Selected_Recipe_Reg_enable D270.04 BOOL  ; On if registration enabled for film
Selected_Recipe_Return_Accel D316 UINT
Selected_Recipe_Return_Decel D317 UINT
Selected_Recipe_Return_Time D314 UINT
Selected_Recipe_Return_Velocity D315 UINT
Selected_Recipe_Rev_Yank_Dist D283 UINT  ; Reverse Yank Distance
Selected_Recipe_Rewind_On_Delay D302 UINT
Selected_Recipe_Seal_Cool D300 UINT
Selected_Recipe_Seal_Delay D298 UINT
Selected_Recipe_Seal_Duration D299 UINT
Selected_Recipe_Spare_Bits_WD0_bit10 D270.10 BOOL  ; Spare
Selected_Recipe_Spare_Bits_WD0_bit11 D270.11 BOOL  ; Spare
Selected_Recipe_Spare_Bits_WD0_bit12 D270.12 BOOL  ; Spare
Selected_Recipe_Spare_Bits_WD0_bit13 D270.13 BOOL  ; Spare
Selected_Recipe_Spare_Bits_WD0_bit14 D270.14 BOOL  ; Spare
Selected_Recipe_Spare_Bits_WD0_bit15 D270.15 BOOL  ; Spare
Selected_Recipe_Spare_Bits_WD0_bit6 D270.06 BOOL  ; Spare
Selected_Recipe_Spare_Bits_WD0_bit7 D270.07 BOOL  ; Spare
Selected_Recipe_Spare_Bits_WD0_bit8 D270.08 BOOL  ; Spare
Selected_Recipe_Spare_Bits_WD0_bit9 D270.09 BOOL  ; Spare
Selected_Recipe_Spare_Bits_WD1_bit0 D271.00 BOOL  ; Spare
Selected_Recipe_Spare_Bits_WD1_bit1 D271.01 BOOL  ; Spare
Selected_Recipe_Spare_Bits_WD1_bit10 D271.10 BOOL  ; Spare
Selected_Recipe_Spare_Bits_WD1_bit11 D271.11 BOOL  ; Spare
Selected_Recipe_Spare_Bits_WD1_bit12 D271.12 BOOL  ; Spare
Selected_Recipe_Spare_Bits_WD1_bit13 D271.13 BOOL  ; Spare
Selected_Recipe_Spare_Bits_WD1_bit14 D271.14 BOOL  ; Spare
Selected_Recipe_Spare_Bits_WD1_bit15 D271.15 BOOL  ; Spare
Selected_Recipe_Spare_Bits_WD1_bit2 D271.02 BOOL  ; Spare
Selected_Recipe_Spare_Bits_WD1_bit3 D271.03 BOOL  ; Spare
Selected_Recipe_Spare_Bits_WD1_bit4 D271.04 BOOL  ; Spare
Selected_Recipe_Spare_Bits_WD1_bit5 D271.05 BOOL  ; Spare
Selected_Recipe_Spare_Bits_WD1_bit6 D271.06 BOOL  ; Spare
Selected_Recipe_Spare_Bits_WD1_bit7 D271.07 BOOL  ; Spare
Selected_Recipe_Spare_Bits_WD1_bit8 D271.08 BOOL  ; Spare
Selected_Recipe_Spare_Bits_WD1_bit9 D271.09 BOOL  ; Spare
Selected_Recipe_Spare_Bits_WD2_bit0 D272.00 BOOL  ; Spare
Selected_Recipe_Spare_Bits_WD2_bit1 D272.01 BOOL  ; Spare
Selected_Recipe_Spare_Bits_WD2_bit10 D272.10 BOOL  ; Spare
Selected_Recipe_Spare_Bits_WD2_bit11 D272.11 BOOL  ; Spare
Selected_Recipe_Spare_Bits_WD2_bit12 D272.12 BOOL  ; Spare
Selected_Recipe_Spare_Bits_WD2_bit13 D272.13 BOOL  ; Spare
Selected_Recipe_Spare_Bits_WD2_bit14 D272.14 BOOL  ; Spare
Selected_Recipe_Spare_Bits_WD2_bit15 D272.15 BOOL  ; Spare
Selected_Recipe_Spare_Bits_WD2_bit2 D272.02 BOOL  ; Spare
Selected_Recipe_Spare_Bits_WD2_bit3 D272.03 BOOL  ; Spare
Selected_Recipe_Spare_Bits_WD2_bit4 D272.04 BOOL  ; Spare
Selected_Recipe_Spare_Bits_WD2_bit5 D272.05 BOOL  ; Spare
Selected_Recipe_Spare_Bits_WD2_bit6 D272.06 BOOL  ; Spare
Selected_Recipe_Spare_Bits_WD2_bit7 D272.07 BOOL  ; Spare
Selected_Recipe_Spare_Bits_WD2_bit8 D272.08 BOOL  ; Spare
Selected_Recipe_Spare_Bits_WD2_bit9 D272.09 BOOL  ; Spare
Selected_Recipe_Spare_Bits_WD3_bit0 D273.00 BOOL  ; Spare
Selected_Recipe_Spare_Bits_WD3_bit1 D273.01 BOOL  ; Spare
Selected_Recipe_Spare_Bits_WD3_bit10 D273.10 BOOL  ; Spare
Selected_Recipe_Spare_Bits_WD3_bit11 D273.11 BOOL  ; Spare
Selected_Recipe_Spare_Bits_WD3_bit12 D273.12 BOOL  ; Spare
Selected_Recipe_Spare_Bits_WD3_bit13 D273.13 BOOL  ; Spare
Selected_Recipe_Spare_Bits_WD3_bit14 D273.14 BOOL  ; Spare
Selected_Recipe_Spare_Bits_WD3_bit15 D273.15 BOOL  ; Spare
Selected_Recipe_Spare_Bits_WD3_bit2 D273.02 BOOL  ; Spare
Selected_Recipe_Spare_Bits_WD3_bit3 D273.03 BOOL  ; Spare
Selected_Recipe_Spare_Bits_WD3_bit4 D273.04 BOOL  ; Spare
Selected_Recipe_Spare_Bits_WD3_bit5 D273.05 BOOL  ; Spare
Selected_Recipe_Spare_Bits_WD3_bit6 D273.06 BOOL  ; Spare
Selected_Recipe_Spare_Bits_WD3_bit7 D273.07 BOOL  ; Spare
Selected_Recipe_Spare_Bits_WD3_bit8 D273.08 BOOL  ; Spare
Selected_Recipe_Spare_Bits_WD3_bit9 D273.09 BOOL  ; Spare
Selected_Recipe_Spare_Bits_WD4_bit0 D274.00 BOOL  ; Spare
Selected_Recipe_Spare_Bits_WD4_bit1 D274.01 BOOL  ; Spare
Selected_Recipe_Spare_Bits_WD4_bit10 D274.10 BOOL  ; Spare
Selected_Recipe_Spare_Bits_WD4_bit11 D274.11 BOOL  ; Spare
Selected_Recipe_Spare_Bits_WD4_bit12 D274.12 BOOL  ; Spare
Selected_Recipe_Spare_Bits_WD4_bit13 D274.13 BOOL  ; Spare
Selected_Recipe_Spare_Bits_WD4_bit14 D274.14 BOOL  ; Spare
Selected_Recipe_Spare_Bits_WD4_bit15 D274.15 BOOL  ; Spare
Selected_Recipe_Spare_Bits_WD4_bit2 D274.02 BOOL  ; Spare
Selected_Recipe_Spare_Bits_WD4_bit3 D274.03 BOOL  ; Spare
Selected_Recipe_Spare_Bits_WD4_bit4 D274.04 BOOL  ; Spare
Selected_Recipe_Spare_Bits_WD4_bit5 D274.05 BOOL  ; Spare
Selected_Recipe_Spare_Bits_WD4_bit6 D274.06 BOOL  ; Spare
Selected_Recipe_Spare_Bits_WD4_bit7 D274.07 BOOL  ; Spare
Selected_Recipe_Spare_Bits_WD4_bit8 D274.08 BOOL  ; Spare
Selected_Recipe_Spare_Bits_WD4_bit9 D274.09 BOOL  ; Spare
Selected_Recipe_Spare_Bits_WD5_bit0 D275.00 BOOL  ; Spare
Selected_Recipe_Spare_Bits_WD5_bit1 D275.01 BOOL  ; Spare
Selected_Recipe_Spare_Bits_WD5_bit10 D275.10 BOOL  ; Spare
Selected_Recipe_Spare_Bits_WD5_bit11 D275.11 BOOL  ; Spare
Selected_Recipe_Spare_Bits_WD5_bit12 D275.12 BOOL  ; Spare
Selected_Recipe_Spare_Bits_WD5_bit13 D275.13 BOOL  ; Spare
Selected_Recipe_Spare_Bits_WD5_bit14 D275.14 BOOL  ; Spare
Selected_Recipe_Spare_Bits_WD5_bit15 D275.15 BOOL  ; Spare
Selected_Recipe_Spare_Bits_WD5_bit2 D275.02 BOOL  ; Spare
Selected_Recipe_Spare_Bits_WD5_bit3 D275.03 BOOL  ; Spare
Selected_Recipe_Spare_Bits_WD5_bit4 D275.04 BOOL  ; Spare
Selected_Recipe_Spare_Bits_WD5_bit5 D275.05 BOOL  ; Spare
Selected_Recipe_Spare_Bits_WD5_bit6 D275.06 BOOL  ; Spare
Selected_Recipe_Spare_Bits_WD5_bit7 D275.07 BOOL  ; Spare
Selected_Recipe_Spare_Bits_WD5_bit8 D275.08 BOOL  ; Spare
Selected_Recipe_Spare_Bits_WD5_bit9 D275.09 BOOL  ; Spare
Selected_Recipe_Spare_Bits_WD6_bit0 D276.00 BOOL  ; Spare
Selected_Recipe_Spare_Bits_WD6_bit1 D276.01 BOOL  ; Spare
Selected_Recipe_Spare_Bits_WD6_bit10 D276.10 BOOL  ; Spare
Selected_Recipe_Spare_Bits_WD6_bit11 D276.11 BOOL  ; Spare
Selected_Recipe_Spare_Bits_WD6_bit12 D276.12 BOOL  ; Spare
Selected_Recipe_Spare_Bits_WD6_bit13 D276.13 BOOL  ; Spare
Selected_Recipe_Spare_Bits_WD6_bit14 D276.14 BOOL  ; Spare
Selected_Recipe_Spare_Bits_WD6_bit15 D276.15 BOOL  ; Spare
Selected_Recipe_Spare_Bits_WD6_bit2 D276.02 BOOL  ; Spare
Selected_Recipe_Spare_Bits_WD6_bit3 D276.03 BOOL  ; Spare
Selected_Recipe_Spare_Bits_WD6_bit4 D276.04 BOOL  ; Spare
Selected_Recipe_Spare_Bits_WD6_bit5 D276.05 BOOL  ; Spare
Selected_Recipe_Spare_Bits_WD6_bit6 D276.06 BOOL  ; Spare
Selected_Recipe_Spare_Bits_WD6_bit7 D276.07 BOOL  ; Spare
Selected_Recipe_Spare_Bits_WD6_bit8 D276.08 BOOL  ; Spare
Selected_Recipe_Spare_Bits_WD6_bit9 D276.09 BOOL  ; Spare
Selected_Recipe_Spare_Bits_WD7_bit0 D277.00 BOOL  ; Spare
Selected_Recipe_Spare_Bits_WD7_bit1 D277.01 BOOL  ; Spare
Selected_Recipe_Spare_Bits_WD7_bit10 D277.10 BOOL  ; Spare
Selected_Recipe_Spare_Bits_WD7_bit11 D277.11 BOOL  ; Spare
Selected_Recipe_Spare_Bits_WD7_bit12 D277.12 BOOL  ; Spare
Selected_Recipe_Spare_Bits_WD7_bit13 D277.13 BOOL  ; Spare
Selected_Recipe_Spare_Bits_WD7_bit14 D277.14 BOOL  ; Spare
Selected_Recipe_Spare_Bits_WD7_bit15 D277.15 BOOL  ; Spare
Selected_Recipe_Spare_Bits_WD7_bit2 D277.02 BOOL  ; Spare
Selected_Recipe_Spare_Bits_WD7_bit3 D277.03 BOOL  ; Spare
Selected_Recipe_Spare_Bits_WD7_bit4 D277.04 BOOL  ; Spare
Selected_Recipe_Spare_Bits_WD7_bit5 D277.05 BOOL  ; Spare
Selected_Recipe_Spare_Bits_WD7_bit6 D277.06 BOOL  ; Spare
Selected_Recipe_Spare_Bits_WD7_bit7 D277.07 BOOL  ; Spare
Selected_Recipe_Spare_Bits_WD7_bit8 D277.08 BOOL  ; Spare
Selected_Recipe_Spare_Bits_WD7_bit9 D277.09 BOOL  ; Spare
Selected_Recipe_Spare_Bits_WD8_bit0 D278.00 BOOL  ; Spare
Selected_Recipe_Spare_Bits_WD8_bit1 D278.01 BOOL  ; Spare
Selected_Recipe_Spare_Bits_WD8_bit10 D278.10 BOOL  ; Spare
Selected_Recipe_Spare_Bits_WD8_bit11 D278.11 BOOL  ; Spare
Selected_Recipe_Spare_Bits_WD8_bit12 D278.12 BOOL  ; Spare
Selected_Recipe_Spare_Bits_WD8_bit13 D278.13 BOOL  ; Spare
Selected_Recipe_Spare_Bits_WD8_bit14 D278.14 BOOL  ; Spare
Selected_Recipe_Spare_Bits_WD8_bit15 D278.15 BOOL  ; Spare
Selected_Recipe_Spare_Bits_WD8_bit2 D278.02 BOOL  ; Spare
Selected_Recipe_Spare_Bits_WD8_bit3 D278.03 BOOL  ; Spare
Selected_Recipe_Spare_Bits_WD8_bit4 D278.04 BOOL  ; Spare
Selected_Recipe_Spare_Bits_WD8_bit5 D278.05 BOOL  ; Spare
Selected_Recipe_Spare_Bits_WD8_bit6 D278.06 BOOL  ; Spare
Selected_Recipe_Spare_Bits_WD8_bit7 D278.07 BOOL  ; Spare
Selected_Recipe_Spare_Bits_WD8_bit8 D278.08 BOOL  ; Spare
Selected_Recipe_Spare_Bits_WD8_bit9 D278.09 BOOL  ; Spare
Selected_Recipe_Spare_UINT0 D333 UINT
Selected_Recipe_Spare_UINT1 D334 UINT
Selected_Recipe_Spare_UINT10 D343 UINT
Selected_Recipe_Spare_UINT100 D433 UINT
Selected_Recipe_Spare_UINT101 D434 UINT
Selected_Recipe_Spare_UINT102 D435 UINT
Selected_Recipe_Spare_UINT103 D436 UINT
Selected_Recipe_Spare_UINT104 D437 UINT
Selected_Recipe_Spare_UINT105 D438 UINT
Selected_Recipe_Spare_UINT106 D439 UINT
Selected_Recipe_Spare_UINT107 D440 UINT
Selected_Recipe_Spare_UINT108 D441 UINT
Selected_Recipe_Spare_UINT109 D442 UINT
Selected_Recipe_Spare_UINT11 D344 UINT
Selected_Recipe_Spare_UINT110 D443 UINT
Selected_Recipe_Spare_UINT111 D444 UINT
Selected_Recipe_Spare_UINT112 D445 UINT
Selected_Recipe_Spare_UINT113 D446 UINT
Selected_Recipe_Spare_UINT114 D447 UINT
Selected_Recipe_Spare_UINT115 D448 UINT
Selected_Recipe_Spare_UINT116 D449 UINT
Selected_Recipe_Spare_UINT117 D450 UINT
Selected_Recipe_Spare_UINT118 D451 UINT
Selected_Recipe_Spare_UINT119 D452 UINT
Selected_Recipe_Spare_UINT12 D345 UINT
Selected_Recipe_Spare_UINT120 D453 UINT
Selected_Recipe_Spare_UINT121 D454 UINT
Selected_Recipe_Spare_UINT122 D455 UINT
Selected_Recipe_Spare_UINT123 D456 UINT
Selected_Recipe_Spare_UINT124 D457 UINT
Selected_Recipe_Spare_UINT125 D458 UINT
Selected_Recipe_Spare_UINT126 D459 UINT
Selected_Recipe_Spare_UINT127 D460 UINT
Selected_Recipe_Spare_UINT128 D461 UINT
Selected_Recipe_Spare_UINT129 D462 UINT
Selected_Recipe_Spare_UINT13 D346 UINT
Selected_Recipe_Spare_UINT130 D463 UINT
Selected_Recipe_Spare_UINT131 D464 UINT
Selected_Recipe_Spare_UINT132 D465 UINT
Selected_Recipe_Spare_UINT133 D466 UINT
Selected_Recipe_Spare_UINT134 D467 UINT
Selected_Recipe_Spare_UINT135 D468 UINT
Selected_Recipe_Spare_UINT136 D469 UINT
Selected_Recipe_Spare_UINT137 D470 UINT
Selected_Recipe_Spare_UINT138 D471 UINT
Selected_Recipe_Spare_UINT139 D472 UINT
Selected_Recipe_Spare_UINT14 D347 UINT
Selected_Recipe_Spare_UINT140 D473 UINT
Selected_Recipe_Spare_UINT141 D474 UINT
Selected_Recipe_Spare_UINT142 D475 UINT
Selected_Recipe_Spare_UINT143 D476 UINT
Selected_Recipe_Spare_UINT144 D477 UINT
Selected_Recipe_Spare_UINT145 D478 UINT
Selected_Recipe_Spare_UINT146 D479 UINT
Selected_Recipe_Spare_UINT147 D480 UINT
Selected_Recipe_Spare_UINT148 D481 UINT
Selected_Recipe_Spare_UINT149 D482 UINT
Selected_Recipe_Spare_UINT15 D348 UINT
Selected_Recipe_Spare_UINT150 D483 UINT
Selected_Recipe_Spare_UINT151 D484 UINT
Selected_Recipe_Spare_UINT152 D485 UINT
Selected_Recipe_Spare_UINT153 D486 UINT
Selected_Recipe_Spare_UINT154 D487 UINT
Selected_Recipe_Spare_UINT155 D488 UINT
Selected_Recipe_Spare_UINT156 D489 UINT
Selected_Recipe_Spare_UINT157 D490 UINT
Selected_Recipe_Spare_UINT158 D491 UINT
Selected_Recipe_Spare_UINT159 D492 UINT
Selected_Recipe_Spare_UINT16 D349 UINT
Selected_Recipe_Spare_UINT160 D493 UINT
Selected_Recipe_Spare_UINT161 D494 UINT
Selected_Recipe_Spare_UINT162 D495 UINT
Selected_Recipe_Spare_UINT163 D496 UINT
Selected_Recipe_Spare_UINT164 D497 UINT
Selected_Recipe_Spare_UINT165 D498 UINT
Selected_Recipe_Spare_UINT166 D499 UINT
Selected_Recipe_Spare_UINT17 D350 UINT
Selected_Recipe_Spare_UINT18 D351 UINT
Selected_Recipe_Spare_UINT19 D352 UINT
Selected_Recipe_Spare_UINT2 D335 UINT
Selected_Recipe_Spare_UINT20 D353 UINT
Selected_Recipe_Spare_UINT21 D354 UINT
Selected_Recipe_Spare_UINT22 D355 UINT
Selected_Recipe_Spare_UINT23 D356 UINT
Selected_Recipe_Spare_UINT24 D357 UINT
Selected_Recipe_Spare_UINT25 D358 UINT
Selected_Recipe_Spare_UINT26 D359 UINT
Selected_Recipe_Spare_UINT27 D360 UINT
Selected_Recipe_Spare_UINT28 D361 UINT
Selected_Recipe_Spare_UINT29 D362 UINT
Selected_Recipe_Spare_UINT3 D336 UINT
Selected_Recipe_Spare_UINT30 D363 UINT
Selected_Recipe_Spare_UINT31 D364 UINT
Selected_Recipe_Spare_UINT32 D365 UINT
Selected_Recipe_Spare_UINT33 D366 UINT
Selected_Recipe_Spare_UINT34 D367 UINT
Selected_Recipe_Spare_UINT35 D368 UINT
Selected_Recipe_Spare_UINT36 D369 UINT
Selected_Recipe_Spare_UINT37 D370 UINT
Selected_Recipe_Spare_UINT38 D371 UINT
Selected_Recipe_Spare_UINT39 D372 UINT
Selected_Recipe_Spare_UINT4 D337 UINT
Selected_Recipe_Spare_UINT40 D373 UINT
Selected_Recipe_Spare_UINT41 D374 UINT
Selected_Recipe_Spare_UINT42 D375 UINT
Selected_Recipe_Spare_UINT43 D376 UINT
Selected_Recipe_Spare_UINT44 D377 UINT
Selected_Recipe_Spare_UINT45 D378 UINT
Selected_Recipe_Spare_UINT46 D379 UINT
Selected_Recipe_Spare_UINT47 D380 UINT
Selected_Recipe_Spare_UINT48 D381 UINT
Selected_Recipe_Spare_UINT49 D382 UINT
Selected_Recipe_Spare_UINT5 D338 UINT
Selected_Recipe_Spare_UINT50 D383 UINT
Selected_Recipe_Spare_UINT51 D384 UINT
Selected_Recipe_Spare_UINT52 D385 UINT
Selected_Recipe_Spare_UINT53 D386 UINT
Selected_Recipe_Spare_UINT54 D387 UINT
Selected_Recipe_Spare_UINT55 D388 UINT
Selected_Recipe_Spare_UINT56 D389 UINT
Selected_Recipe_Spare_UINT57 D390 UINT
Selected_Recipe_Spare_UINT58 D391 UINT
Selected_Recipe_Spare_UINT59 D392 UINT
Selected_Recipe_Spare_UINT6 D339 UINT
Selected_Recipe_Spare_UINT60 D393 UINT
Selected_Recipe_Spare_UINT61 D394 UINT
Selected_Recipe_Spare_UINT62 D395 UINT
Selected_Recipe_Spare_UINT63 D396 UINT
Selected_Recipe_Spare_UINT64 D397 UINT
Selected_Recipe_Spare_UINT65 D398 UINT
Selected_Recipe_Spare_UINT66 D399 UINT
Selected_Recipe_Spare_UINT67 D400 UINT
Selected_Recipe_Spare_UINT68 D401 UINT
Selected_Recipe_Spare_UINT69 D402 UINT
Selected_Recipe_Spare_UINT7 D340 UINT
Selected_Recipe_Spare_UINT70 D403 UINT
Selected_Recipe_Spare_UINT71 D404 UINT
Selected_Recipe_Spare_UINT72 D405 UINT
Selected_Recipe_Spare_UINT73 D406 UINT
Selected_Recipe_Spare_UINT74 D407 UINT
Selected_Recipe_Spare_UINT75 D408 UINT
Selected_Recipe_Spare_UINT76 D409 UINT
Selected_Recipe_Spare_UINT77 D410 UINT
Selected_Recipe_Spare_UINT78 D411 UINT
Selected_Recipe_Spare_UINT79 D412 UINT
Selected_Recipe_Spare_UINT8 D341 UINT
Selected_Recipe_Spare_UINT80 D413 UINT
Selected_Recipe_Spare_UINT81 D414 UINT
Selected_Recipe_Spare_UINT82 D415 UINT
Selected_Recipe_Spare_UINT83 D416 UINT
Selected_Recipe_Spare_UINT84 D417 UINT
Selected_Recipe_Spare_UINT85 D418 UINT
Selected_Recipe_Spare_UINT86 D419 UINT
Selected_Recipe_Spare_UINT87 D420 UINT
Selected_Recipe_Spare_UINT88 D421 UINT
Selected_Recipe_Spare_UINT89 D422 UINT
Selected_Recipe_Spare_UINT9 D342 UINT
Selected_Recipe_Spare_UINT90 D423 UINT
Selected_Recipe_Spare_UINT91 D424 UINT
Selected_Recipe_Spare_UINT92 D425 UINT
Selected_Recipe_Spare_UINT93 D426 UINT
Selected_Recipe_Spare_UINT94 D427 UINT
Selected_Recipe_Spare_UINT95 D428 UINT
Selected_Recipe_Spare_UINT96 D429 UINT
Selected_Recipe_Spare_UINT97 D430 UINT
Selected_Recipe_Spare_UINT98 D431 UINT
Selected_Recipe_Spare_UINT99 D432 UINT
Selected_Recipe_Stale_Film_Time D329 UINT
Selected_Recipe_Temp_Setpoint D281 UINT  ; Tool temperature setpoint
Selected_Recipe_Tool_Position D319 UINT
Selected_Recipe_Top_Vacuum_Delay D286 UINT
Selected_Recipe_Tray_Position D313 UINT
Selected_Recipe_Tray_Settle_Time D307 UINT
Selected_Recipe_Tray_Stop_Delay D304 UINT
Selected_Recipe_Upstream_Off_Delay D312 UINT
Selected_Recipe_Upstream_On_Delay D311 UINT
Selected_Recipe_VAC_Type D270.00 BOOL  ; Vac type - ON = Pressure, OFF = Time
Selected_Recipe_Vacuum_Duration D288 UINT
Selected_Recipe_Vacuum_Extra_Time D290 UINT
Selected_Recipe_Vacuum_Pressure_SP D289 UINT
Selected_Recipe_Vent_Bottom_Delay D295 UINT
Selected_Recipe_Vent_Bottom_Duration D296 UINT
Selected_Recipe_Vent_Pressure_SP D297 UINT
Selected_Recipe_Vent_Top_Delay D294 UINT
Selected_Recipe_Vent_Type D270.02 BOOL  ; Vent type - ON = Pressure, OFF = Time
Servo_Drive_OK 2960.01 BOOL  ; The servo drive has no error
Servo_Drive_Reset 2961.05 BOOL  ; Reset output to servo drive
Servo_Fault W150.14 BOOL  ; Servo drive fault
Servo_Home_OK W497.01 BOOL  ; Servo home has been initiated after power up or estop condition.
Servo_On_Machine W202.15 BOOL  ; The machine has a servo drive
Simultaneous_Mode W201.04 BOOL
Sleep_Mode W151.11 BOOL  ; Sleep Mode enabled - drop temp and fault
Sleep_Mode_Delay T0220 TIMER  ; Delay to Start Sleep mode
Sleep_Mode_Minutes D898 UINT
Sleep_Mode_Temperature D899 UINT
Sleep_Mode_Temporary_Value D1142 UINT  ; Temporary register to hold the temperature setpoint while in sleep mode
Sleep_Time_SP D1140 DINT  ; Sleep timer setpoint
Slow_Down_DIstance D2400 DINT
Slow_Down_Decel H162 DINT
Slow_Down_Speed_Frequency H163 DINT  ; H163/164
Slow_Vent_Delay T0143 TIMER  ; Delay for Slow Vent
Stale_Film_timer T0215 TIMER  ; Stale film
Start_Status D800 UINT  ; Indicator status for start PB
Stepper_Pulse_Output A281.04 BOOL  ; Pulses are being output
Stop_Command W202.05 BOOL
Stop_Latch W202.04 BOOL
Stop_Status D801 UINT  ; Indicator status for stop PB
TC1_Temp_Fdbk T0150 TIMER  ; TC1 Temp Feedback Fault Delay
TC2_Temp_Fdbk T0151 TIMER  ; TC2 Temp Feedback Fault Delay
TC_AT_Enabled W501.08 BOOL  ; Set when Auto Tune is enabled
TC_Global_AT W501.06 BOOL  ; TC Global Auto Tune
TC_Loop1_AT W500.01 BOOL  ; Auto Tune Loop1
TC_Loop2_AT W500.02 BOOL  ; Auto Tune Loop2
TC_Loop3_AT W500.03 BOOL  ; Auto Tune Loop3
TC_Loop4_AT W500.04 BOOL  ; Auto Tune Loop4
TC_Loop5_AT W500.05 BOOL  ; Auto Tune Loop5
TC_Loop6_AT W500.06 BOOL  ; Auto Tune Loop6
TC_MOD1_Feedback_Fault W151.08 BOOL  ; TC Module 1 RTD Feedback Fault
TC_MOD2_Feedback_Fault W151.09 BOOL  ; TC module 2 RTD Feedback Fault
TC_PID_PROM W501.07 BOOL  ; Save PID to TC EEPROM
TC_PID_Recipe W501.10 BOOL  ; Move PID to recipe when saving
TPM D803 UINT  ; Trays Per Minute
TPO_Control_Period_Heater1 D6044 UINT  ; Time in 0.01s units of control period (200 = 2.00 seconds)
TPO_Control_Period_Heater2 D6094 UINT  ; Time in 0.01s units of control period (200 = 2.00 seconds)
TPO_Control_Period_Heater3 D6144 UINT  ; Time in 0.01s units of control period (200 = 2.00 seconds)
TPO_Control_Period_Heater4 D6194 UINT  ; Time in 0.01s units of control period (200 = 2.00 seconds)
TPO_Control_Period_Heater5 D6244 UINT  ; Time in 0.01s units of control period (200 = 2.00 seconds)
TPO_Out_Lower_Limit_Heater1 D6045 UINT  ; TPO Output lower limit when enabled in D5100.
TPO_Out_Lower_Limit_Heater2 D6095 UINT  ; TPO Output lower limit when enabled in D6043.
TPO_Out_Lower_Limit_Heater3 D6145 UINT  ; TPO Output lower limit when enabled in D6043.
TPO_Out_Lower_Limit_Heater4 D6195 UINT  ; TPO Output lower limit when enabled in D6043.
TPO_Out_Lower_Limit_Heater5 D6245 UINT  ; TPO Output lower limit when enabled in D6043.
TPO_Out_Upper_Limit_Heater1 D6046 UINT  ; TPO Output Upper limit when enabled in D5043.
TPO_Out_Upper_Limit_Heater2 D6096 UINT  ; TPO Output Upper limit when enabled in D6100.
TPO_Out_Upper_Limit_Heater3 D6146 UINT  ; TPO Output Upper limit when enabled in D6100.
TPO_Out_Upper_Limit_Heater4 D6196 UINT  ; TPO Output Upper limit when enabled in D6100.
TPO_Out_Upper_Limit_Heater5 D6246 UINT  ; TPO Output Upper limit when enabled in D6100.
TPO_Parameter1_Heater1 D6043 CHANNEL  ; Sets output limit function, input read timing, input type and MV Range
TPO_Parameter1_Heater2 D6093 CHANNEL  ; Sets output limit function, input read timing, input type and MV Range
TPO_Parameter1_Heater3 D6143 CHANNEL  ; Sets output limit function, input read timing, input type and MV Range
TPO_Parameter1_Heater4 D6193 CHANNEL  ; Sets output limit function, input read timing, input type and MV Range
TPO_Parameter1_Heater5 D6243 CHANNEL  ; Sets output limit function, input read timing, input type and MV Range
TPO_Percent_Heater1 D6042 UINT  ; Percentage output from PIDAT function
TPO_Percent_Heater2 D6092 UINT  ; Percentage output from PIDAT function
TPO_Percent_Heater3 D6142 UINT  ; Percentage output from PIDAT function
TPO_Percent_Heater4 D6192 UINT  ; Percentage output from PIDAT function
TPO_Percent_Heater5 D6242 UINT  ; Percentage output from PIDAT function
TPO_Work_Area_Word1_Heater1 D6047 CHANNEL  ; TPO Work Area - DO NOT USE FOR ANYTHING ELSE
TPO_Work_Area_Word1_Heater2 D6097 CHANNEL  ; TPO Work Area - DO NOT USE FOR ANYTHING ELSE
TPO_Work_Area_Word1_Heater3 D6147 CHANNEL  ; TPO Work Area - DO NOT USE FOR ANYTHING ELSE
TPO_Work_Area_Word1_Heater4 D6197 CHANNEL  ; TPO Work Area - DO NOT USE FOR ANYTHING ELSE
TPO_Work_Area_Word1_Heater5 D6247 CHANNEL  ; TPO Work Area - DO NOT USE FOR ANYTHING ELSE
TPO_Work_Area_Word2_Heater1 D6048 CHANNEL  ; TPO Work Area - DO NOT USE FOR ANYTHING ELSE
TPO_Work_Area_Word2_Heater2 D6098 CHANNEL  ; TPO Work Area - DO NOT USE FOR ANYTHING ELSE
TPO_Work_Area_Word2_Heater3 D6148 CHANNEL  ; TPO Work Area - DO NOT USE FOR ANYTHING ELSE
TPO_Work_Area_Word2_Heater4 D6198 CHANNEL  ; TPO Work Area - DO NOT USE FOR ANYTHING ELSE
TPO_Work_Area_Word2_Heater5 D6248 CHANNEL  ; TPO Work Area - DO NOT USE FOR ANYTHING ELSE
TPO_Work_Area_Word3_Heater1 D6049 CHANNEL  ; TPO Work Area - DO NOT USE FOR ANYTHING ELSE
TPO_Work_Area_Word3_Heater2 D6099 CHANNEL  ; TPO Work Area - DO NOT USE FOR ANYTHING ELSE
TPO_Work_Area_Word3_Heater3 D6149 CHANNEL  ; TPO Work Area - DO NOT USE FOR ANYTHING ELSE
TPO_Work_Area_Word3_Heater4 D6199 CHANNEL  ; TPO Work Area - DO NOT USE FOR ANYTHING ELSE
TPO_Work_Area_Word3_Heater5 D6249 CHANNEL  ; TPO Work Area - DO NOT USE FOR ANYTHING ELSE
Temp1_Feedback_disconnected 2009.04 BOOL  ; Input Signal Disconnected
Temp2Conv C_to_F
Temp2_Feedback_disconnected 2009.05 BOOL  ; Input Signal disconnected
Temp3Conv C_to_F
Temp4Conv C_to_F
Temp5Conv C_to_F
Temp_AutoTune_Heater1 D6009.15 BOOL  ; Initiates Autotune function
Temp_AutoTune_Heater2 D6059.15 BOOL  ; Initiates Autotune function
Temp_AutoTune_Heater3 D6109.15 BOOL  ; Initiates Autotune function
Temp_AutoTune_Heater4 D6159.15 BOOL  ; Initiates Autotune function
Temp_AutoTune_Heater5 D6209.15 BOOL  ; Initiates Autotune function
Temp_Derivative_Constant_Heater1 D6003 UINT  ; Derivative constant - 0.1s units &0 means not used
Temp_Derivative_Constant_Heater2 D6053 UINT  ; Derivative constant - 0.1s units &0 means not used
Temp_Derivative_Constant_Heater3 D6103 UINT  ; Derivative constant - 0.1s units &0 means not used
Temp_Derivative_Constant_Heater4 D6153 UINT  ; Derivative constant - 0.1s units &0 means not used
Temp_Derivative_Constant_Heater5 D6203 UINT  ; Derivative constant - 0.1s units &0 means not used
Temp_Integral_Constant_Heater1 D6002 UINT  ; Integral constant - 0.1s units.  &9999 means not used
Temp_Integral_Constant_Heater2 D6052 UINT  ; Integral constant - 0.1s units.  &9999 means not used
Temp_Integral_Constant_Heater3 D6102 UINT  ; Integral constant - 0.1s units.  &9999 means not used
Temp_Integral_Constant_Heater4 D6152 UINT  ; Integral constant - 0.1s units.  &9999 means not used
Temp_Integral_Constant_Heater5 D6202 UINT  ; Integral constant - 0.1s units.  &9999 means not used
Temp_Limit_Cycle_Hysteresis_Heater1 D6010 UINT  ; Hysteresis for limit cycle
Temp_Limit_Cycle_Hysteresis_Heater2 D6060 UINT  ; Hysteresis for limit cycle
Temp_Limit_Cycle_Hysteresis_Heater3 D6110 UINT  ; Hysteresis for limit cycle
Temp_Limit_Cycle_Hysteresis_Heater4 D6160 UINT  ; Hysteresis for limit cycle
Temp_Limit_Cycle_Hysteresis_Heater5 D6210 UINT  ; Hysteresis for limit cycle
Temp_Prop_band_Heater1 D6001 UINT  ; Proportional band in 0.1% units
Temp_Prop_band_Heater2 D6051 UINT  ; Proportional band in 0.1% units
Temp_Prop_band_Heater3 D6101 UINT  ; Proportional band in 0.1% units
Temp_Prop_band_Heater4 D6151 UINT  ; Proportional band in 0.1% units
Temp_Prop_band_Heater5 D6201 UINT  ; Proportional band in 0.1% units
Temp_Sampling_period_Heater1 D6004 UINT  ; Sampling period 0.01s units.
Temp_Sampling_period_Heater2 D6054 UINT  ; Sampling period 0.01s units.
Temp_Sampling_period_Heater3 D6104 UINT  ; Sampling period 0.01s units.
Temp_Sampling_period_Heater4 D6154 UINT  ; Sampling period 0.01s units.
Temp_Sampling_period_Heater5 D6204 UINT  ; Sampling period 0.01s units.
Temp_Set_Value_Heater1 D6000 UINT  ; Set value for the PIDAT Function
Temp_Set_Value_Heater2 D6050 UINT  ; Set value for the PIDAT Function
Temp_Set_Value_Heater3 D6100 UINT  ; Set value for the PIDAT Function
Temp_Set_Value_Heater4 D6150 UINT  ; Set value for the PIDAT Function
Temp_Set_Value_Heater5 D6200 UINT  ; Set value for the PIDAT Function
Temperature_Pressure_Scale Conv_Scale_analog_with_Int_range
Teperature_Low W150.13 BOOL  ; Temperature not high enough to run product
Termperature_High W151.07 BOOL  ; Temperature too high enough to run product
Tool_Close_Decel_Delay_Timer T0113 TIMER  ; Tool Close Delay
Tool_Down_Prox 0.03 BOOL  ; Tool down proximity sw
Tool_Down_Timer T0202 TIMER  ; Time to hold decel before releasing
Tool_Lift_Down_Decel_manual W200.05 BOOL  ; Manual tool lift down decel command
Tool_Lift_Up_Decel_manual W200.04 BOOL  ; Manual tool lift up decel command
Tool_Not_Clamped_Fault W151.04 BOOL  ; The Upper Tool Is Not Locked
Tool_Open_Decel_Delay_Timer T0112 TIMER  ; Tool Open delay
Tool_Position_HMIx10 D876 DINT
Tool_Up_Prox 0.02 BOOL  ; Tool up proximity sw
Tool_clamp_memory D967 UINT
Transducer_Fault W151.10 BOOL  ; Transducer disconnected
Tray1_AT_On_Flag 2028.03 BOOL  ; Loop1 Auto Tune ON
Tray1_ChangePIDConstants 2022.13 BOOL  ; Loop1 Turn Off PID constant flag
Tray1_Constants_Calculated 2028.10 BOOL  ; Loop1 PID Constants Calc flag
Tray1_ControlPeriod_SP D20213 UINT
Tray1_Derivative D20217 UINT
Tray1_FATALCONTROL_Error 2028.12 BOOL  ; Loop1 FATAL CONTROL Error
Tray1_Integral_Time D20216 UINT
Tray1_Output_On 2028.04 BOOL  ; Loop1 Control Output ON
Tray1_PID_Save 2022.15 BOOL  ; Loop1 Save to EEPROM
Tray1_PV 2023 INT  ; Loop1 Process Value
Tray1_Proportional D20215 UINT
Tray1_SENSOR_Error 2028.14 BOOL  ; Loop1 SENSOR error
Tray1_SETTING_Error 2028.09 BOOL  ; Loop1 SETTING Error
Tray1_SP 2020 INT  ; Loop1 Setpoint
Tray1_Save_Complete 2028.15 BOOL  ; Loop1 Save to EEPROM complete
Tray1_Start_AT 2022.02 BOOL  ; Loop1 Start Auto Tune
Tray1_Stop 2022.06 BOOL  ; Loop1 Stop Controlling
Tray1_StopAT 2022.03 BOOL  ; Loop1 Stop Auto Tune
Tray1_Stop_Sensor 1.00 BOOL  ; Tray stop sensor input
Tray1_Temp_Fdbk T0145 TIMER  ; Tray 1 Temp Feedback Fault Delay
Tray1and2_Alarm_Mode D20200 CHANNEL
Tray2_AT_On_Flag 2029.03 BOOL  ; Loop2 Auto Tune ON
Tray2_ChangePIDConstants 2022.12 BOOL  ; Loop2 Turn Off PID constant flag
Tray2_Constants_Calculated 2029.10 BOOL  ; Loop2 PID Constants Calc flag
Tray2_ControlPeriod_SP D20223 UINT
Tray2_Derivative D20227 UINT
Tray2_FATALCONTROL_Error 2029.12 BOOL  ; Loop2 FATAL CONTROL Error
Tray2_Integral_Time D20226 UINT
Tray2_Output_On 2029.04 BOOL  ; Loop2 Control Output ON
Tray2_PID_Save 2022.14 BOOL  ; Loop2 Save to EEPROM
Tray2_PV 2024 INT  ; Loop2 Process Value
Tray2_Proportional D20225 UINT
Tray2_SENSOR_Error 2029.14 BOOL  ; Loop2 SENSOR error
Tray2_SETTING_Error 2029.09 BOOL  ; Loop2 SETTING Error
Tray2_SP 2021 INT  ; Loop2 Setpoint
Tray2_Save_Complete 2029.15 BOOL  ; Loop2 Save to EEPROM complete
Tray2_Start_AT 2022.00 BOOL  ; Loop2 Start Auto Tune
Tray2_Stop 2022.04 BOOL  ; Loop2 Stop Controlling
Tray2_Stop_AT 2022.01 BOOL  ; Loop2 Stop Auto Tune
Tray2_Stop_Sensor 1.01 BOOL  ; Tray stop sensor input
Tray2_Temp_Fdbk T0146 TIMER  ; Tray 2 Temp Feedback Fault Delay
Tray3_AT_On_Flag 2038.03 BOOL  ; Loop3 Auto Tune ON
Tray3_ChangePIDConstants 2032.13 BOOL  ; Loop3 Turn Off PID constant flag
Tray3_Constants_Calculated 2038.10 BOOL  ; Loop3 PID Constants Calc flag
Tray3_ControlPeriod_SP D20253 UINT
Tray3_Derivative D20257 UINT
Tray3_FATALCONTROL_Error 2038.12 BOOL  ; Loop3 FATAL CONTROL Error
Tray3_Integral_Time D20256 UINT
Tray3_Output_On 2038.04 BOOL  ; Loop3 Control Output ON
Tray3_PID_Save 2032.15 BOOL  ; Loop3 Save to EEPROM
Tray3_PV 2033 INT  ; Loop3 Process Value
Tray3_Proportional D20255 UINT
Tray3_SENSOR_Error 2038.14 BOOL  ; Loop3 SENSOR error
Tray3_SETTING_Error 2038.09 BOOL  ; Loop3 SETTING Error
Tray3_SP 2030 INT  ; Loop 3 Setpoint
Tray3_Save_Complete 2038.15 BOOL  ; Loop3 Save to EEPROM complete
Tray3_Start_AT 2032.02 BOOL  ; Loop3 Start Auto Tune
Tray3_Stop 2032.06 BOOL  ; Loop3 Stop Controlling
Tray3_Stop_AT 2032.03 BOOL  ; Loop3 Stop Auto Tune
Tray3_Stop_Sensor 1.02 BOOL  ; Tray stop sensor input
Tray3_Temp_Fdbk T0147 TIMER  ; Tray 3 Temp Feedback Fault Delay
Tray3and4_Alarm_Mode D20201 CHANNEL
Tray4_AT_On_Flag 2039.03 BOOL  ; Loop4 Auto Tune ON
Tray4_ChangePIDConstants 2032.12 BOOL  ; Loop4 Turn Off PID constant flag
Tray4_Constants_Calculated 2039.10 BOOL  ; Loop4 PID Constants Calc flag
Tray4_ControlPeriod_SP D20263 UINT
Tray4_Derivative D20267 UINT
Tray4_FATALCONTROL_Error 2039.12 BOOL  ; Loop4 FATAL CONTROL Error
Tray4_Integral_Time D20266 UINT
Tray4_Output_On 2039.04 BOOL  ; Loop4 Control Output ON
Tray4_PID_Save 2032.14 BOOL  ; Loop4 Save to EEPROM
Tray4_PV 2034 INT  ; Loop4 Process Value
Tray4_Proportional D20265 UINT
Tray4_SENSOR_Error 2039.14 BOOL  ; Loop4 SENSOR error
Tray4_SETTING_Error 2039.09 BOOL  ; Loop4 SETTING Error
Tray4_SP 2031 INT  ; Loop 4 Setpoint
Tray4_Save_Complete 2039.15 BOOL  ; Loop4 Save to EEPROM complete
Tray4_Start_AT 2032.00 BOOL  ; Loop4 Start Auto Tune
Tray4_Stop 2032.04 BOOL  ; Loop4 Stop Controlling
Tray4_Stop_AT 2032.01 BOOL  ; Loop4 Stop Auto Tune
Tray4_Stop_Sensor 1.03 BOOL  ; Tray stop sensor input
Tray4_Temp_Fdbk T0148 TIMER  ; Tray 4 Temp Feedback Fault Delay
Tray5_AT_On_Flag 2128.03 BOOL  ; Loop5 Auto Tune ON
Tray5_ChangePIDConstants 2122.13 BOOL  ; Loop5 Turn Off PID constant flag
Tray5_Constants_Calculated 2128.10 BOOL  ; Loop5 PID Constants Calc flag
Tray5_ControlPeriod_SP D21213 UINT
Tray5_Derivative D21217 UINT
Tray5_FATALCONTROL_Error 2128.12 BOOL  ; Loop5 FATAL CONTROL Error
Tray5_Integral_Time D21216 UINT
Tray5_Output_On 2128.04 BOOL  ; Loop5 Control Output ON
Tray5_PID_Save 2122.15 BOOL  ; Loop5 Save to EEPROM
Tray5_PV 2123 INT  ; Loop5 Process Value
Tray5_Proportional D21215 UINT
Tray5_SENSOR_Error 2128.14 BOOL  ; Loop5 SENSOR error
Tray5_SETTING_Error 2128.09 BOOL  ; Loop5 SETTING Error
Tray5_SP 2120 INT  ; Loop 5 Setpoint
Tray5_Save_Complete 2128.15 BOOL  ; Loop5 Save to EEPROM complete
Tray5_Start_AT 2122.02 BOOL  ; Loop5 Start Auto Tune
Tray5_Stop 2122.06 BOOL  ; Loop5 Stop Controlling
Tray5_StopAT 2122.03 BOOL  ; Loop5 Stop Auto Tune
Tray5_Stop_Sensor 1.04 BOOL  ; Tray stop sensor input
Tray5_Temp_Fdbk T0149 TIMER  ; Tray 5 Temp Feedback Fault Delay
Tray5and6_Alarm_Mode D21200 CHANNEL
Tray6_ControlPeriod_SP D21223 UINT
Tray6_Derivative D21227 UINT
Tray6_Integral_Time D21226 UINT
Tray6_Proportional D21225 UINT
TrayCountChanged W203.08 BOOL  ; The tray count has been changed.
TrayStop1_Off_Filter_Timer T0262 TIMER
TrayStop2_Off_Filter_Timer T0263 TIMER
TrayStop3_Off_Filter_Timer T0264 TIMER
TrayStop4_Off_Filter_Timer T0265 TIMER
TrayStop5_Off_Filter_Timer T0266 TIMER
TrayStop6_Off_Filter_Timer T0267 TIMER
Tray_Count D512 UINT  ; Trays past the infeed gate
Tray_Detected_4_measurement 1.09 BOOL  ; Photocell to detect trays for measurement
Tray_Height_Int D2026 UINT  ; Tray height in INT form
Tray_Height_memory1 D2027 UINT  ; Measured hieght of tray 1
Tray_Height_memory2 D2028 UINT  ; Measured height of tray2
Tray_Height_memory3 D2029 UINT  ; Measured height of tray3
Tray_Height_memory4 D2030 UINT  ; Measured height of tray4
Tray_Height_memory5 D2031 UINT  ; Measured height of tray5
Tray_Measured T0242 TIMER  ; Measured Time for tray passage
Tray_Measurement_bits D2034 UINT  ; Bits used for tray measurement
Tray_Measurement_counter D2033 UINT  ; Measurement counter
Tray_Position_HMIx10 D878 DINT
Tray_count_TPM D965 UINT
Tray_filter T0253 TIMER  ; Filter signal for tray counting
Tray_measure_delay T0251 TIMER  ; Delay tray measurement
Tray_measurement_bits D2034.00 BOOL  ; Meaurement in progress
Tray_measurement_temp D2032 UINT  ; temporary memory location for tray height
Tray_measurement_timer T0252 TIMER  ; Time to measure tray
UPPER_TOOL_UNLOCK_DELAY T0126 TIMER  ; Delay Upper Tool from Unlocking
UnitRestart_TC102_1 A502.02 BOOL  ; Restart TC102 Module 1
UnitRestart_TC102_2 A502.12 BOOL  ; Restart TC102 Module 2
UpStream_Conv_Timer_Input T0224 TIMER  ; UpStream_Conv_Timer_Input_HMI
UpStream_Conv_photo_Eye 1.08 BOOL  ; UpStream Conv. Photo-Eye
UpperTool_Unlocked_Status H100.00 BOOL
Upper_Tool_DN_EStop W203.12 BOOL  ; Send Upper Tool Down if E-Stop hit during Lock motion
Upper_Tool_Feedback_NOP W203.14 BOOL
Upper_Tool_Jammed W153.13 BOOL  ; Upper Tool Jammed while trying to close
Upper_Tool_Lock_WD_Fault W150.06 BOOL  ; Watchdog Timer Fault
Upper_Tool_Lock_WD_Timer T0135 TIMER  ; Watchdog Timer
Upper_Tool_Locked W203.09 BOOL  ; Upper Tool Locked when a Safety Faults
Upper_Tool_NOT_Locked W203.11 BOOL  ; Upper Tool NOT Locked Bit
Upper_Tool_Pressure 2005 UINT  ; Upper Tool Pressure
Upper_Tool_Temp_IN5 2017 UINT
Upper_Tool_UNLocked W203.10 BOOL  ; Upper Tool UnLocked when a Safety Trips
Upper_Tool_Unlock_WD_Fault W150.07 BOOL  ; Watchdog Timer Fault
Upper_Tool_Unlock_WD_Timer T0136 TIMER  ; Watchdog Timer
Upper_Tool_Unlocked H100.00 BOOL  ; Upper Tool unlocked status
Upper_Tool_Up_Request W203.13 BOOL  ; HMI Tool Up/Lock Pressed
Upper_Vac_Duration_Simultaneous_Timer T0208 TIMER  ; Used for simultaneous Mode
Upstream_Off_Timer T0210 TIMER  ; OFF Delay timer for upstream signal
Upstream_On_Timer T0209 TIMER  ; ON Delay timer for upstream signal
V10_Tray_2_Stop_Extend 3.09 BOOL  ; V10 Tray Stop 2 Extend output
V11_Tray_Stop3_Extend 4.03 BOOL  ; V11 Tray Stop 3 Extend output
V12_Tray_Stop4_Extend 4.04 BOOL  ; V12 Tray Stop 4 Extend output
V13_Tray_Stop5_Extend 4.05 BOOL  ; V13 Tray Stop 5 Extend output
V14_Infeed_Gate_Retract 3.04 BOOL  ; V14 Infeed Gate Retract output
V15A_Seal_Bar_Retract 2.06 BOOL  ; V15A Seal Bar Retract output
V15B_Seal_Bars_Extend 2.07 BOOL  ; V15B Seal Bar Extend output
V16A_Lower_Tool_Up 2.14 BOOL  ; V16A Lower Tool Lift Up output
V16B_Lower_Tool_Dn 2.15 BOOL  ; V16B Lower Tool Lift Down output
V17A_Lower_Tool_Up_Decel 3.00 BOOL  ; V17A Lower Tool Decel for Up movement
V17B_Lower_Tool_Dn_Decel 3.01 BOOL  ; V17B Lower Tool Decel for Down movement
V1A_Upper_Tool_Vac 2.09 BOOL  ; V1A Upper Tool Vac On output
V1B_Upper_Tool_Vent_Close 2.10 BOOL  ; V1B Upper Tool Vent Close output
V2A_Lower_Tool_Vac 2.11 BOOL  ; V2A Lower Tool Vacuum On output
V2B_Lower_Tool_Vent_Close 2.12 BOOL  ; V2B Vent Close On output
V33_Upstream_Tray_Stop 3.13 BOOL  ; V33 Upstream_Conv_Tray_Stop
V4A_Gripper_Close 3.02 BOOL  ; V4A Tray Gripper Close output
V4B_Gripper_Open 3.03 BOOL  ; V4B Tray Gripper Open output
V5A_Gas_On 2.13 BOOL  ; V5A Gas ON output
V5B_Slow_Top_Vent 3.12 BOOL  ; V5B Slow Top Vent -Option
V6A_Upper_Tool_UnLock 2.03 BOOL  ; V6A Unlock Upper Tool Seat
V6B_Upper_Tool_Lock 3.11 BOOL  ; V6B Lock/Raise Upper Tool-double solenoid valve only
V7_Lower_Tool_Center_Seal 2.04 BOOL  ; V7 Lower Tool Center Seal On
V8A_Gripper_Extend 3.05 BOOL  ; V8A Gripper Extend output-IN450 ONLY
V8B_Gripper_Retract 3.06 BOOL  ; V8B Gripper Retract output-IN450 ONLY
V9_Tray_1_Stop_Extend 3.08 BOOL  ; V9 Tray 1 Stop 1 Extend output
VSP_Mode W201.05 BOOL
VacGraph_Pause W503.02 BOOL  ; graph pause
Vac_Delay_Timer_Bottom T0115 TIMER  ; Vacuum delay timer -Bottom Valve
Vac_Delay_Timer_Top T0114 TIMER  ; Vacuum delay timer - Top Valve
Vac_Duration_Timer T0116 TIMER  ; Vacuum duration
Vac_Test1 Vac_Test_Calc
Vac_Test_Cycle_Timer T0218 TIMER  ; Allowable time for cycle
Vac_Test_Leak_Time D1138 CHANNEL  ; Time for pressure to leak off
Vac_Test_Leak_reached W202.03 BOOL  ; The leak pressure has been reached.
Vac_Test_Pressure_Reached W202.02 BOOL  ; Vacuum test pressure reached
Vac_Test_Result_Time D1137 UINT  ; Time to draw vacuum
Vac_Test_Vent_Timer T0217 TIMER  ; Vent timer release for vacuum test
Vac_Test_ended_early W202.07 BOOL  ; Vac test ended early
Vac_Timeout_WD_Fault W150.05 BOOL  ; Watchdog Timer Fault
Vac_Timeout_WD_Timer T0134 TIMER  ; Watchdog Timer
Vacuum_Extra_time T0219 TIMER
Vacuum_Pump_OK 0.14 BOOL  ; Vacuum pump OK input
Vacuum_Test_Fault W151.06 BOOL
Vacuum_Test_Finished W203.05 BOOL  ; Vacuum test completely finished
Vacuum_Test_Status D960 UINT
Vent_Delay_Timer_Bottom T0120 TIMER  ; Vent Delay Timer - Bottom Valve
Vent_Delay_Timer_Top T0119 TIMER  ; Vent Delay Timer - Top Valve
Vent_Duration_Timer T0121 TIMER  ; Vent duration Timer
Vent_Timeout_WD_Fault W150.10 BOOL  ; Watchdog Timer Fault
Vent_Timeout_WD_Timer T0139 TIMER  ; Watchdog Timer
Vx_UpStream_Tray_Stop_Extend 4.06 BOOL  ; Vx Upstream Conveyor Tray Stop Extend
Yank_Accel_Rate H20 UINT
Yank_Decel_Rate H21 UINT
Yank_Distance_Negative D1114 DINT
Yank_Starting_Freq H26 DINT
Yank_Target_Frequency H22 DINT
Yank_Target_Position H24 DINT
aiCard2_Channel4 2018 UINT
aiForceEnable_Card1Channel4 D2010.05 BOOL  ; unused
aiForceEnable_UpperToolTemp1 D2010.02 BOOL  ; Temperature input1 upper tool force enable
aiForceEnable_UpperToolTemp2 D2010.03 BOOL  ; Temperature input2 upper tool force enable
aiForceEnable_VacuumPressure D2010.04 BOOL  ; pressure transducer for upper tool force enable
aiValue_Card1Channel4 D2025 UINT  ; unused
aiValue_UpperToolTemp1 D2022 UINT  ; Temperature input1 upper tool logical value
aiValue_UpperToolTemp2 D2023 UINT  ; Temperature input2 upper tool logical value
aiValue_VacuumPressure D2024 UINT  ; pressure transducer for upper tool logical value
aoForceEnable_Card1Channel2 D2010.01 BOOL  ; One shot for Measure
aoForceEnable_InfeedConveyorSpeedRef D2010.00 BOOL  ; Analog output for speed reference force enable
aoValue_Card1Channel2 D2021 UINT  ; unused
aoValue_InfeedConveyorSpeedRef D2020 UINT  ; Analog output for speed reference logical value
bActivateSealBarHeating D5053.00 BOOL
bEnglishMode D910.00 BOOL
bFaultOverTemperature D5053.01 BOOL
bFaultTemperatureDeviation D5053.02 BOOL
bGripperJogCommanded D5053.09 BOOL  ; jog button pressed on HMI
bGripperJogging D5053.10 BOOL  ; gripper in jog sequence
bSetTempControlParameters D5053.04 BOOL
bTunePID D5053.03 BOOL
cfgAi1MeanSampleSetting D20006 CHANNEL  ; set to 16 samples for mean
cfgAi2MeanSampleSetting D20007 CHANNEL  ; set to 16 samples for mean
cfgAi3MeanSampleSetting D20008 CHANNEL  ; set to 8 samples for mean
cfgAi4MeanSampleSetting D20009 CHANNEL  ; set to 8 samples for mean
gas_rescale_result D2045 WORD
iGripperJogStep D5500 UINT
iTempDeviationHolder D5055 UINT
iTempDeviationHolder1 D5057 UINT
ipCard2Bit10 1.10 BOOL  ; unused
ipForceEnable_ACDrive_OK D2002.07 BOOL  ; AC Drive Input Force enable
ipForceEnable_AirPressureOk D2000.04 BOOL  ; Air Pressure switch Force enable
ipForceEnable_FrontGrippedClosed D2000.07 BOOL  ; Front Gripper closed proximity sw Force enable
ipForceEnable_FrontGripperOpen D2000.06 BOOL  ; Front Gripper open proximity switch Force enable
ipForceEnable_GasPressureOk D2000.05 BOOL  ; Gas Pressure Switch Force enable
ipForceEnable_GripperExtended D2000.08 BOOL  ; Gripper extended proximity sw Force enable
ipForceEnable_GripperRetracted D2000.09 BOOL  ; Gripper retracted proximity sw Force enable
ipForceEnable_GuardAuthority D2000.15 BOOL  ; Guard Authority input Force enable
ipForceEnable_GuardOk D2000.11 BOOL  ; Guard door switches ok Force enable
ipForceEnable_InfeedEstop D2000.01 BOOL  ; E-Stop circuit status Force enable
ipForceEnable_InfeedGate D2000.12 BOOL  ; Infeed Gate Sensor Force enable
ipForceEnable_OutfeedEstop D2000.10 BOOL  ; E-Stop circuit status Force enable
ipForceEnable_Rear_Gripper_Closed_Prox D2002.06 BOOL  ; Rear Gripper closed prox Force Enable
ipForceEnable_Rear_Gripper_Open_Prox D2002.05 BOOL  ; Rear Gripper Open prox Force Enable
ipForceEnable_RemotePause D2000.13 BOOL  ; Remote pause input Force enable
ipForceEnable_RewindDancerUp D2000.00 BOOL  ; Proximity sw input Force enable
ipForceEnable_StopSensorTray1 D2002.00 BOOL  ; Tray stop sensor input Force enable
ipForceEnable_StopSensorTray2 D2002.01 BOOL  ; Tray stop sensor input Force enable
ipForceEnable_StopSensorTray3 D2002.02 BOOL  ; Tray stop sensor input Force enable
ipForceEnable_StopSensorTray4 D2002.03 BOOL  ; Tray stop sensor input Force enable
ipForceEnable_StopSensorTray5 D2002.04 BOOL  ; Tray stop sensor input Force enable
ipForceEnable_ToolDown D2000.03 BOOL  ; Tool down proximity sw Force enable
ipForceEnable_ToolUp D2000.02 BOOL  ; Tool up proximity sw Force enable
ipForceEnable_VacuumPumpOk D2000.14 BOOL  ; Vacuum pump OK input Force enable
ipForceEnable_ipCard2Bit10 D2002.10 BOOL  ; unused Force enable
ipForceEnable_ipCard2Bit11 D2002.11 BOOL  ; unused Force enable
ipForceEnable_ipCard2Bit12 D2002.12 BOOL  ; unused Force enable
ipForceEnable_ipCard2Bit13 D2002.13 BOOL  ; unused Force enable
ipForceEnable_ipCard2Bit14 D2002.14 BOOL  ; unused Force enable
ipForceEnable_ipCard2Bit15 D2002.15 BOOL  ; unused Force enable
ipForceEnable_ipCard2Bit7 D2002.07 BOOL  ; unused Force enable
ipForceEnable_ipCard2Bit8 D2002.08 BOOL  ; unused Force enable
ipForceEnable_ipCard2Bit9 D2002.09 BOOL  ; unused Force enable
ipState_AC_Drive_OK D2003.07 BOOL  ; AC Drive OK input logical State
ipState_AirPressureOk D2001.04 BOOL  ; Air Pressure switch logical State
ipState_FrontGrippedClosed D2001.07 BOOL  ; Front Gripper closed proximity sw logical State
ipState_FrontGripperOpen D2001.06 BOOL  ; Front Gripper open proximity switch logical State
ipState_GasPressureOk D2001.05 BOOL  ; Gas Pressure Switch logical State
ipState_GripperExtended D2001.08 BOOL  ; Gripper extended proximity sw logical State
ipState_GripperRetracted D2001.09 BOOL  ; Gripper retracted proximity sw logical State
ipState_GuardAuthority D2001.15 BOOL  ; Guard Authority input logical State
ipState_GuardOk D2001.11 BOOL  ; Guard door switches ok logical State
ipState_InfeedEstop D2001.01 BOOL  ; E-Stop circuit status logical State
ipState_InfeedGate D2001.12 BOOL  ; Infeed Gate Sensor logical State
ipState_OutfeedEstop D2001.10 BOOL  ; E-Stop circuit status logical State
ipState_Printer_Fault D2003.15 BOOL  ; Bell-Mark Printer
ipState_Printer_Ready D2003.14 BOOL  ; Bell-Mark Printer
ipState_Rear_Gripper_Closed_Prox D2003.06 BOOL  ; Rear gripper closed logical state
ipState_Rear_Gripper_Open_Prox D2003.05 BOOL  ; Rear gripper Open logical state
ipState_RemotePause D2001.13 BOOL  ; Remote pause input logical State
ipState_RewindDancerUp D2001.00 BOOL  ; Proximity sw input logical State
ipState_StopSensorTray1 D2003.00 BOOL  ; Tray stop sensor input logical State
ipState_StopSensorTray2 D2003.01 BOOL  ; Tray stop sensor input logical State
ipState_StopSensorTray3 D2003.02 BOOL  ; Tray stop sensor input logical State
ipState_StopSensorTray4 D2003.03 BOOL  ; Tray stop sensor input logical State
ipState_StopSensorTray5 D2003.04 BOOL  ; Tray stop sensor input logical State
ipState_ToolDown D2001.03 BOOL  ; Tool down proximity sw logical State
ipState_ToolUp D2001.02 BOOL  ; Tool up proximity sw logical State
ipState_UpStream_PE D2003.08 BOOL  ; UpStream_Photo_Eye
ipState_VacuumPumpOk D2001.14 BOOL  ; Vacuum pump OK input logical State
ipState_ipCard2Bit10 D2003.10 BOOL  ; unused logical State
ipState_ipCard2Bit11 D2003.11 BOOL  ; Infeed safety door
ipState_ipCard2Bit12 D2003.12 BOOL  ; Front or Back Door Safety
ipState_ipCard2Bit13 D2003.13 BOOL
ipState_ipCard2Bit9 D2003.09 BOOL  ; unused logical State
keyswitch_Input_Access 1.12 BOOL  ; Keyswitc input for access to parameters
opCard2Bit14 3.14 BOOL  ; unused
opCard3Bit10 4.10 BOOL  ; unused
opCard3Bit11 4.11 BOOL  ; unused
opCard3Bit12 4.12 BOOL  ; unused
opCard3Bit13 4.13 BOOL  ; unused
opCard3Bit7 4.07 BOOL  ; unused
opCard3Bit8 4.08 BOOL  ; unused
opCard3Bit9 4.09 BOOL  ; unused
opForceEnable_Card2Bit12 D2006.12 BOOL  ; unused Force enable
opForceEnable_Card2Bit13 D2006.13 BOOL  ; unused Force enable
opForceEnable_Card2Bit14 D2006.14 BOOL  ; unused Force enable
opForceEnable_Card2Bit15 D2006.15 BOOL  ; unused Force enable
opForceEnable_Card3Bit10 D2008.10 BOOL  ; unused Force enable
opForceEnable_Card3Bit11 D2008.11 BOOL  ; unused Force enable
opForceEnable_Card3Bit12 D2008.12 BOOL  ; unused Force enable
opForceEnable_Card3Bit13 D2008.13 BOOL  ; unused Force enable
opForceEnable_Card3Bit7 D2008.07 BOOL  ; unused Force enable
opForceEnable_Card3Bit8 D2008.08 BOOL  ; unused Force enable
opForceEnable_Card3Bit9 D2008.09 BOOL  ; unused Force enable
opForceEnable_GasOn D2004.13 BOOL  ; Gas ON output Force enable
opForceEnable_GripperExtend D2006.05 BOOL  ; Gripper Extend output Force enable
opForceEnable_GripperRetract D2006.06 BOOL  ; Gripper Retract output Force enable
opForceEnable_HeatCR D2004.00 BOOL  ; Heat contactor output Force enable
opForceEnable_InfeedConveyorRun D2006.07 BOOL  ; Run the infeed conveyor Force enable
opForceEnable_InfeedGateRetract D2006.04 BOOL  ; Infeed gate retract output Force enable
opForceEnable_LowerToolLiftDown D2004.15 BOOL  ; Lower tool lift down output Force enable
opForceEnable_LowerToolLiftDownDecel D2006.01 BOOL  ; Tool Decel output for down movement Force enable
opForceEnable_LowerToolLiftUp D2004.14 BOOL  ; Lower tool lift up output Force enable
opForceEnable_LowerToolLiftUpDecel D2006.00 BOOL  ; Tool Decel output for up movement Force enable
opForceEnable_LowerToolVac D2004.11 BOOL  ; Lower tool vacuum output Force enable
opForceEnable_LowerToolVentClose D2004.12 BOOL  ; Vent close output Force enable
opForceEnable_Printer_Enable D2008.14 BOOL  ; Bell-Mark Printer
opForceEnable_Printer_Print D2008.15 BOOL  ; Bell-Mark Printer
opForceEnable_RewindMotorStarter D2004.08 BOOL  ; Rewind Motor output Force enable
opForceEnable_SealBarExtend D2004.07 BOOL  ; Seal bars extend output Force enable
opForceEnable_SealBarHeat D2004.01 BOOL  ; Seal Bar Heat output Force enable
opForceEnable_SealBarHeat_2 D2004.02 BOOL  ; Seal Bar Heat output logical State Heater 2
opForceEnable_SealBarRetract D2004.06 BOOL  ; Seal bar retract output Force enable
opForceEnable_Seal_Bar_Heat_3 D2008.00 BOOL  ; Seal Bar Heat output 3 Force Enable
opForceEnable_Seal_Bar_Heat_4 D2008.01 BOOL  ; Seal Bar Heat output 4 Force Enable
opForceEnable_Seal_Bar_Heat_5 D2008.02 BOOL  ; Seal Bar Heat output 5 Force Enable
opForceEnable_TrayGripClose D2006.02 BOOL  ; Grip close output Force enable
opForceEnable_TrayGripOpen D2006.03 BOOL  ; Grip open output Force enable
opForceEnable_TrayStop1Extend D2006.08 BOOL  ; Tray stop 1 extend output Force enable
opForceEnable_TrayStop2Extend D2006.09 BOOL  ; Tray stop 2 extend output Force enable
opForceEnable_Tray_Stop3_Extend D2008.03 BOOL  ; Tray stop 3 extend output Force Enable
opForceEnable_Tray_Stop4_Extend D2008.04 BOOL  ; Tray stop 4 extend output Force Enable
opForceEnable_Tray_Stop5_Extend D2008.05 BOOL  ; Tray stop 5 extend output Force Enable
opForceEnable_UpperToolVac D2004.09 BOOL  ; Upper tool vacuum output Force enable
opForceEnable_UpperToolVentClose D2004.10 BOOL  ; Upper tool vent close output Force enable
opForceEnable_UpstreamStop D2006.10 BOOL  ; Upstream Stop output Force enable
opForceEnable_V6A_UpperToolSeat D2004.03 BOOL  ; V6A Upper Tool Seat UNLock Force enable
opForceEnable_V6B_UpperTool_Lock D2006.11 BOOL  ; Upper Tool Lock Output Force enable
opForceEnable_V7_LowerToolSeal D2004.04 BOOL  ; V7 Lower tool Center Seal output Force enable
opForceEnable_VacuumPump D2004.05 BOOL  ; Vacuum Pump output Force enable
opForceState_V6UpperToolSeat W102.05 BOOL  ; used to force Upper Tool seat output
opForceUpstream_Stop D2008.06 BOOL  ; Force Enable for upstream stop
opState_Card2Bit14 D2007.14 BOOL  ; unused logical State
opState_Force_Tool_Decel_Down D2009.08 BOOL  ; Force Decel Down Immediately
opState_GasOn D2005.13 BOOL  ; Gas ON output logical State
opState_GripperExtend D2007.05 BOOL  ; Gripper Extend output logical State
opState_GripperRetract D2007.06 BOOL  ; Gripper Retract output logical State
opState_HeatCR D2005.00 BOOL  ; Heat contactor output logical State
opState_InfeedConveyorRun D2007.07 BOOL  ; Run the infeed conveyor logical State
opState_InfeedGateRetract D2007.04 BOOL  ; Infeed gate retract output logical State
opState_Lift_Up_B4_lowering D2009.09 BOOL  ; Reenergize Lift before lowering
opState_LowerToolLiftDown D2005.15 BOOL  ; Lower tool lift down output logical State
opState_LowerToolLiftDownDecel D2007.01 BOOL  ; Tool Decel output for down movement logical State
opState_LowerToolLiftUp D2005.14 BOOL  ; Lower tool lift up output logical State
opState_LowerToolLiftUpDecel D2007.00 BOOL  ; Tool Decel output for up movement logical State
opState_LowerToolVac D2005.11 BOOL  ; Lower tool vacuum output logical State
opState_LowerToolVentClose D2005.12 BOOL  ; Vent close output logical State
opState_Outfeed_Conveyor D2007.15 BOOL  ; Run outfeed conveyor
opState_Printer_Enable D2009.14 BOOL  ; Bell-Mark Printer
opState_Printer_Print D2009.15 BOOL  ; Bell-Mark Printer
opState_Renergize_button D2009.10 BOOL  ; HMI open and exit button
opState_RewindMotorStarter D2005.08 BOOL  ; Rewind Motor output logical State
opState_SealBar1_Heat D2005.01 BOOL  ; Seal Bar 1 Heat output logical State
opState_SealBarExtend D2005.07 BOOL  ; Seal bars extend output logical State
opState_SealBarRetract D2005.06 BOOL  ; Seal bar retract output logical State
opState_Seal_Bar_Heat_3 D2009.00 BOOL  ; Seal Bar Heat output 3
opState_Seal_Bar_Heat_4 D2009.01 BOOL  ; Seal Bar Heat output 4
opState_Seal_Bar_Heat_5 D2009.02 BOOL  ; Seal Bar Heat output 5
opState_Sealbar2_heat D2005.02 BOOL  ; Heat output for seal bar 2
opState_TrayGripClose D2007.02 BOOL  ; Grip close output logical State
opState_TrayGripOpen D2007.03 BOOL  ; Grip open output logical State
opState_TrayStop1Extend D2007.08 BOOL  ; Tray stop 1 extend output logical State
opState_TrayStop2Extend D2007.09 BOOL  ; Tray stop 2 extend output logical State
opState_TrayStop3Extend D2009.03 BOOL  ; Extend Tray stop 3
opState_TrayStop4Extend D2009.04 BOOL  ; Extend tray stop 4
opState_TrayStop5Extend D2009.05 BOOL  ; Extend tray stop 5
opState_UpperToolVac D2005.09 BOOL  ; Upper tool vacuum output logical State
opState_UpperToolVentClose D2005.10 BOOL  ; Upper tool vent close output logical State
opState_UpstreamStop D2007.10 BOOL  ; Upstream Stop output logical State
opState_Upstream_Stop_Bit_2 D2009.07 BOOL  ; Upstream Stop bit
opState_V33_Upstream_Stop D2007.13 BOOL  ; V33 Upstream Conv Stop logical State
opState_V5B_Slow_Top_Vent D2007.12 BOOL  ; V5B Slow Top Vent TEST
opState_V6A_UpperTool_Lock D2005.03 BOOL  ; V6A Upper Tool Seat UNLock logical State
opState_V6B_Upper_Tool_Lock D2007.11 BOOL  ; V6B Upper Tool Lock logical State
opState_V7LowerToolSeal D2005.04 BOOL  ; V7 Lower tool Center Seal output logical State
opState_VacuumPump D2005.05 BOOL  ; Vacuum Pump output logical State
opState_reenergize_up_B4_lowering D2009.09 BOOL  ; reenergize the lift before dropping
op_State_Upstream_Stop_TYSON D2009.06 BOOL  ; Logical state for upstream stop-TYSONS Only
over_run D2034.01 BOOL
tray_measurement T0240 TIMER  ; Tray measure at infeed gate
tray_measurement2 T0241 TIMER  ; Tray Measure at stop 3

## Program Main (cyclic task 0)
Local symbols
ipState_InFeed_Gaurd 2003.11 BOOL  ; Infeed safety door

### Section Startup

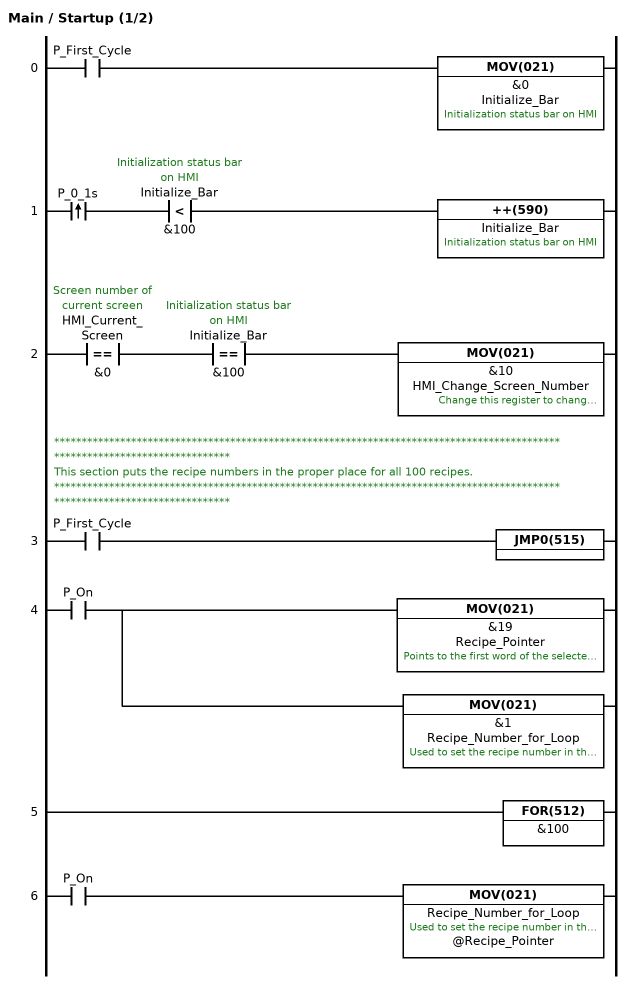
; rung 0
LD P_First_Cycle
MOV(021) &0 Initialize_Bar  ; Initialization status bar on HMI
; rung 1
@LD P_0_1s
AND<(310) Initialize_Bar &100  ; Initialization status bar on HMI
++(590) Initialize_Bar  ; Initialization status bar on HMI
; rung 2
LD=(300) HMI_Current_Screen &0  ; Screen number of current screen
AND=(300) Initialize_Bar &100  ; Initialization status bar on HMI
MOV(021) &10 HMI_Change_Screen_Number  ; Change this register to change screens
; rung 3: **************************************************************************************************************************** / This section puts the recipe numbers in the proper place for all 100 recipes. / ****************************************************************************************************************************
LD P_First_Cycle
JMP0(515)
; rung 4
LD P_On
MOV(021) &19 Recipe_Pointer  ; Points to the first word of the selected recipe in the recipe memory area (E0 - E24999)
MOV(021) &1 Recipe_Number_for_Loop  ; Used to set the recipe number in the recipe tables
; rung 5
FOR(512) &100
; rung 6
LD P_On
MOV(021) Recipe_Number_for_Loop @Recipe_Pointer  ; Used to set the recipe number in the recipe tables

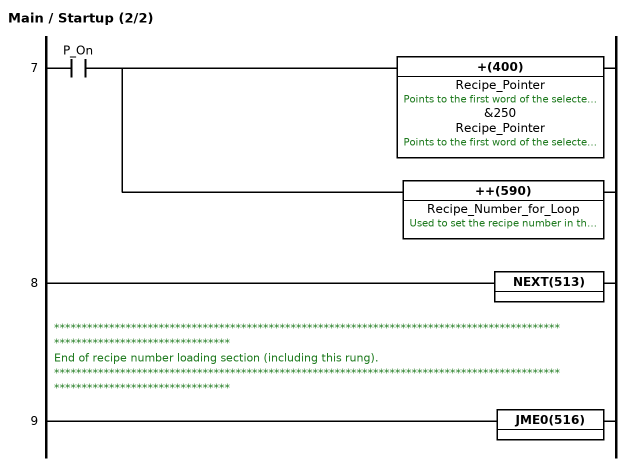
; rung 7
LD P_On
+(400) Recipe_Pointer &250 Recipe_Pointer  ; Points to the first word of the selected recipe in the recipe memory area (E0 - E24999)
++(590) Recipe_Number_for_Loop  ; Used to set the recipe number in the recipe tables
; rung 8
NEXT(513)
; rung 9: **************************************************************************************************************************** / End of recipe number loading section (including this rung). / ****************************************************************************************************************************
JME0(516)

### Section Recipe_Handling

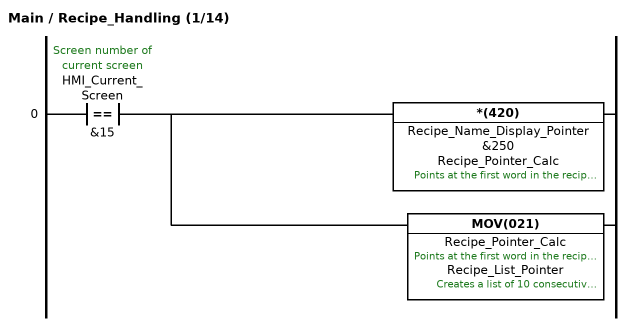
; rung 0
LD=(300) HMI_Current_Screen &15  ; Screen number of current screen
*(420) Recipe_Name_Display_Pointer &250 Recipe_Pointer_Calc  ; Points at the first word in the recipe storage area (E0 - E24999) for the selected recipe.
MOV(021) Recipe_Pointer_Calc Recipe_List_Pointer  ; Points at the first word in the recipe storage area (E0 - E24999) for the selected recipe., Creates a list of 10 consecutive recipe names

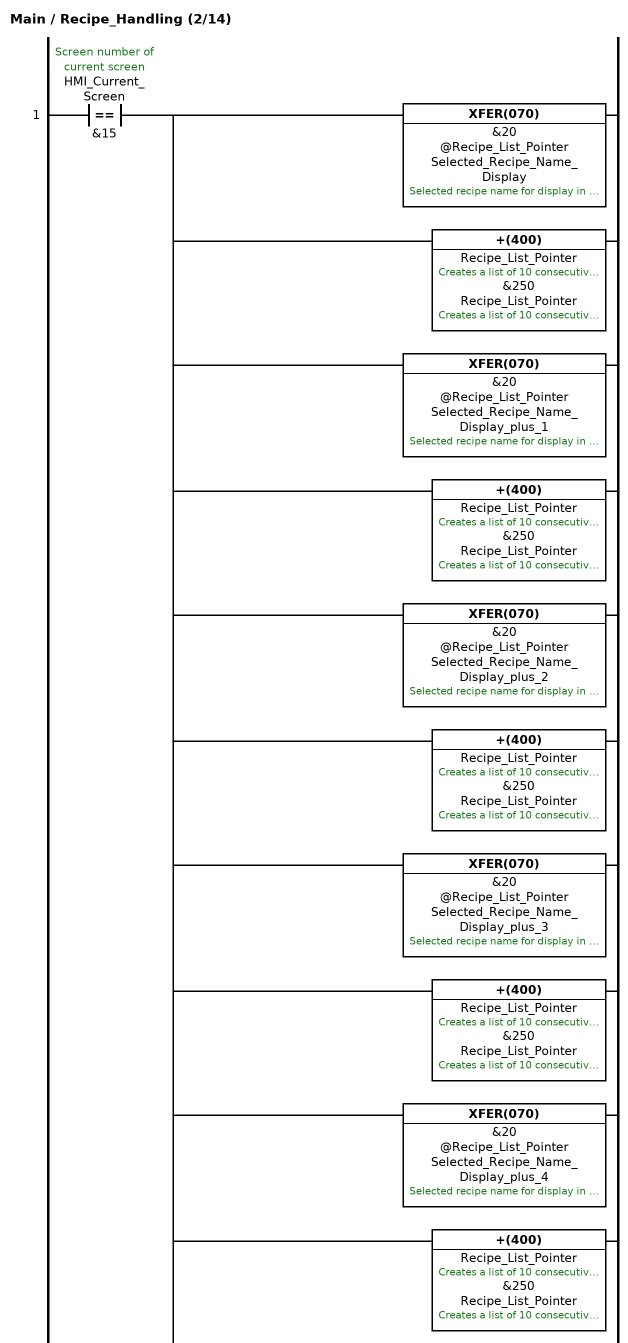

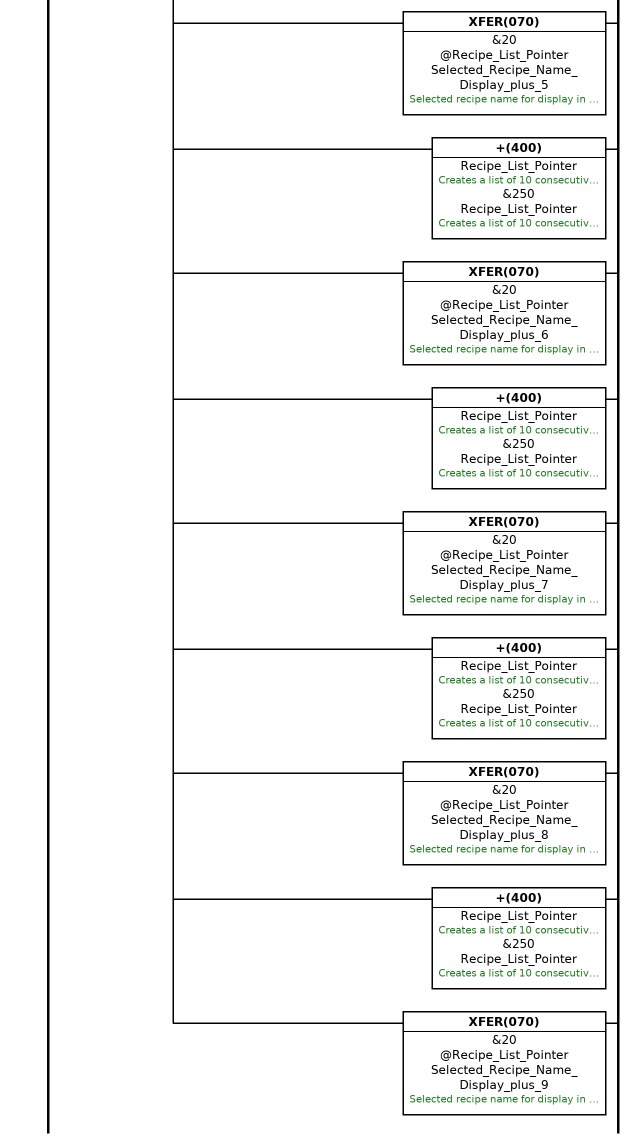
; rung 1
LD=(300) HMI_Current_Screen &15  ; Screen number of current screen
XFER(070) &20 @Recipe_List_Pointer Selected_Recipe_Name_Display  ; Selected recipe name for display in a list.
+(400) Recipe_List_Pointer &250 Recipe_List_Pointer  ; Creates a list of 10 consecutive recipe names
XFER(070) &20 @Recipe_List_Pointer Selected_Recipe_Name_Display_plus_1  ; Selected recipe name for display in a list.  Selected + 1
+(400) Recipe_List_Pointer &250 Recipe_List_Pointer  ; Creates a list of 10 consecutive recipe names
XFER(070) &20 @Recipe_List_Pointer Selected_Recipe_Name_Display_plus_2  ; Selected recipe name for display in a list.  Selected + 2
+(400) Recipe_List_Pointer &250 Recipe_List_Pointer  ; Creates a list of 10 consecutive recipe names
XFER(070) &20 @Recipe_List_Pointer Selected_Recipe_Name_Display_plus_3  ; Selected recipe name for display in a list.  Selected + 3
+(400) Recipe_List_Pointer &250 Recipe_List_Pointer  ; Creates a list of 10 consecutive recipe names
XFER(070) &20 @Recipe_List_Pointer Selected_Recipe_Name_Display_plus_4  ; Selected recipe name for display in a list.  Selected + 4
+(400) Recipe_List_Pointer &250 Recipe_List_Pointer  ; Creates a list of 10 consecutive recipe names
XFER(070) &20 @Recipe_List_Pointer Selected_Recipe_Name_Display_plus_5  ; Selected recipe name for display in a list.  Selected + 5
+(400) Recipe_List_Pointer &250 Recipe_List_Pointer  ; Creates a list of 10 consecutive recipe names
XFER(070) &20 @Recipe_List_Pointer Selected_Recipe_Name_Display_plus_6  ; Selected recipe name for display in a list.  Selected + 6
+(400) Recipe_List_Pointer &250 Recipe_List_Pointer  ; Creates a list of 10 consecutive recipe names
XFER(070) &20 @Recipe_List_Pointer Selected_Recipe_Name_Display_plus_7  ; Selected recipe name for display in a list.  Selected + 7
+(400) Recipe_List_Pointer &250 Recipe_List_Pointer  ; Creates a list of 10 consecutive recipe names
XFER(070) &20 @Recipe_List_Pointer Selected_Recipe_Name_Display_plus_8  ; Selected recipe name for display in a list.  Selected + 8
+(400) Recipe_List_Pointer &250 Recipe_List_Pointer  ; Creates a list of 10 consecutive recipe names
XFER(070) &20 @Recipe_List_Pointer Selected_Recipe_Name_Display_plus_9  ; Selected recipe name for display in a list.  Selected + 9

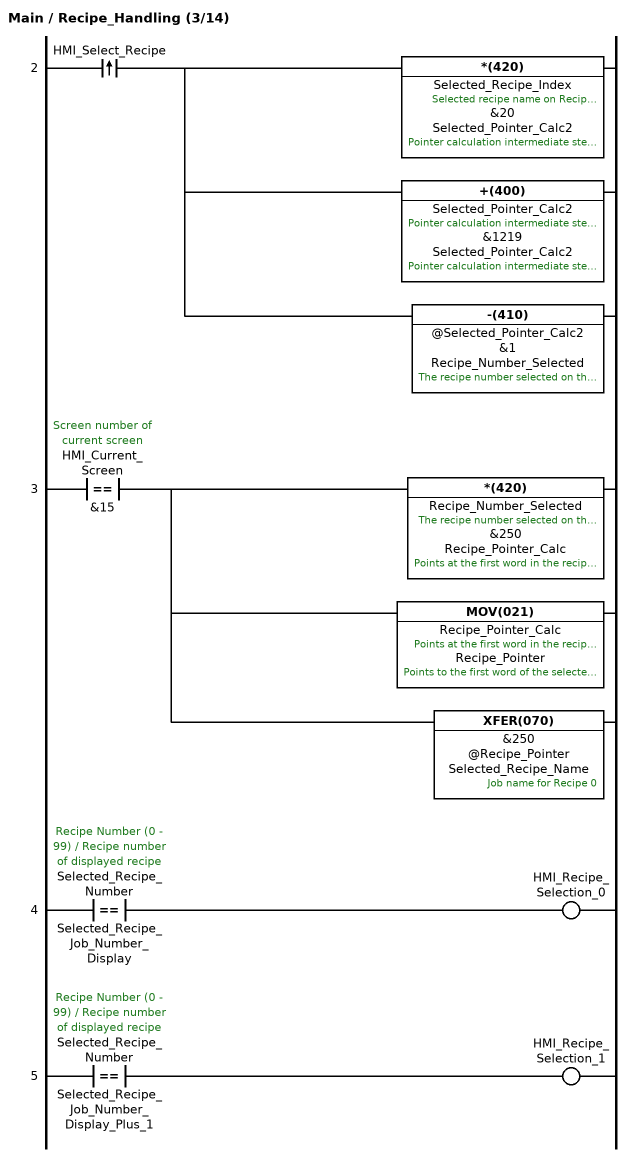
; rung 2
@LD HMI_Select_Recipe
*(420) Selected_Recipe_Index &20 Selected_Pointer_Calc2  ; Selected recipe name on Recipe Screen, Pointer calculation intermediate step 2
+(400) Selected_Pointer_Calc2 &1219 Selected_Pointer_Calc2  ; Pointer calculation intermediate step 2
-(410) @Selected_Pointer_Calc2 &1 Recipe_Number_Selected  ; The recipe number selected on the screen.
; rung 3
LD=(300) HMI_Current_Screen &15  ; Screen number of current screen
*(420) Recipe_Number_Selected &250 Recipe_Pointer_Calc  ; The recipe number selected on the screen., Points at the first word in the recipe storage area (E0 - E24999) for the selected recipe.
MOV(021) Recipe_Pointer_Calc Recipe_Pointer  ; Points at the first word in the recipe storage area (E0 - E24999) for the selected recipe., Points to the first word of the selected recipe in the recipe memory area (E0 - E24999)
XFER(070) &250 @Recipe_Pointer Selected_Recipe_Name  ; Job name for Recipe 0
; rung 4
LD=(300) Selected_Recipe_Number Selected_Recipe_Job_Number_Display  ; Recipe Number (0 - 99), Recipe number of displayed recipe
OUT HMI_Recipe_Selection_0
; rung 5
LD=(300) Selected_Recipe_Number Selected_Recipe_Job_Number_Display_Plus_1  ; Recipe Number (0 - 99), Recipe number of displayed recipe
OUT HMI_Recipe_Selection_1

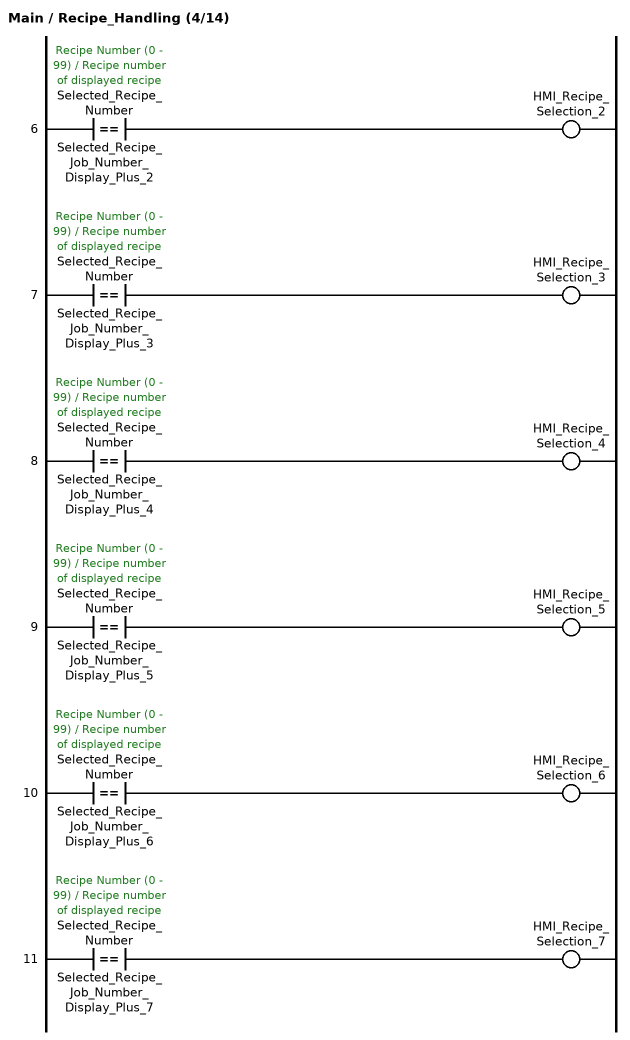
; rung 6
LD=(300) Selected_Recipe_Number Selected_Recipe_Job_Number_Display_Plus_2  ; Recipe Number (0 - 99), Recipe number of displayed recipe
OUT HMI_Recipe_Selection_2
; rung 7
LD=(300) Selected_Recipe_Number Selected_Recipe_Job_Number_Display_Plus_3  ; Recipe Number (0 - 99), Recipe number of displayed recipe
OUT HMI_Recipe_Selection_3
; rung 8
LD=(300) Selected_Recipe_Number Selected_Recipe_Job_Number_Display_Plus_4  ; Recipe Number (0 - 99), Recipe number of displayed recipe
OUT HMI_Recipe_Selection_4
; rung 9
LD=(300) Selected_Recipe_Number Selected_Recipe_Job_Number_Display_Plus_5  ; Recipe Number (0 - 99), Recipe number of displayed recipe
OUT HMI_Recipe_Selection_5
; rung 10
LD=(300) Selected_Recipe_Number Selected_Recipe_Job_Number_Display_Plus_6  ; Recipe Number (0 - 99), Recipe number of displayed recipe
OUT HMI_Recipe_Selection_6
; rung 11
LD=(300) Selected_Recipe_Number Selected_Recipe_Job_Number_Display_Plus_7  ; Recipe Number (0 - 99), Recipe number of displayed recipe
OUT HMI_Recipe_Selection_7

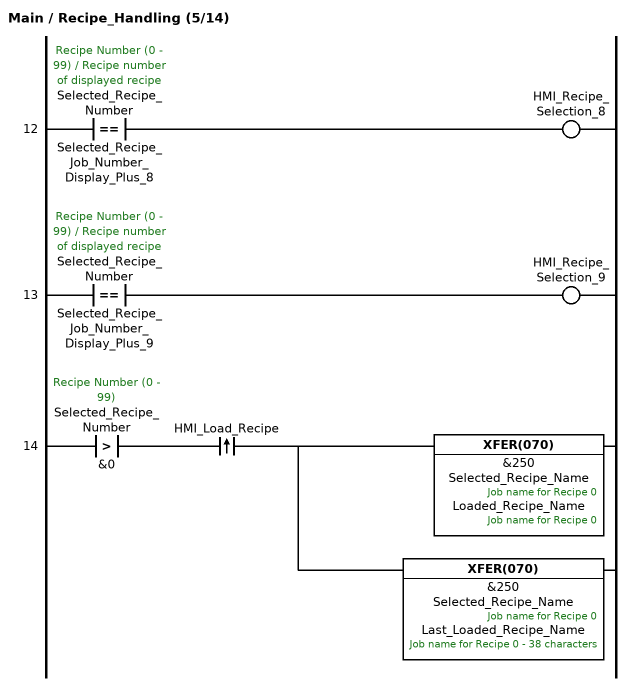
; rung 12
LD=(300) Selected_Recipe_Number Selected_Recipe_Job_Number_Display_Plus_8  ; Recipe Number (0 - 99), Recipe number of displayed recipe
OUT HMI_Recipe_Selection_8
; rung 13
LD=(300) Selected_Recipe_Number Selected_Recipe_Job_Number_Display_Plus_9  ; Recipe Number (0 - 99), Recipe number of displayed recipe
OUT HMI_Recipe_Selection_9
; rung 14
LD>(320) Selected_Recipe_Number &0  ; Recipe Number (0 - 99)
@AND HMI_Load_Recipe
XFER(070) &250 Selected_Recipe_Name Loaded_Recipe_Name  ; Job name for Recipe 0
XFER(070) &250 Selected_Recipe_Name Last_Loaded_Recipe_Name  ; Job name for Recipe 0, Job name for Recipe 0 - 38 characters

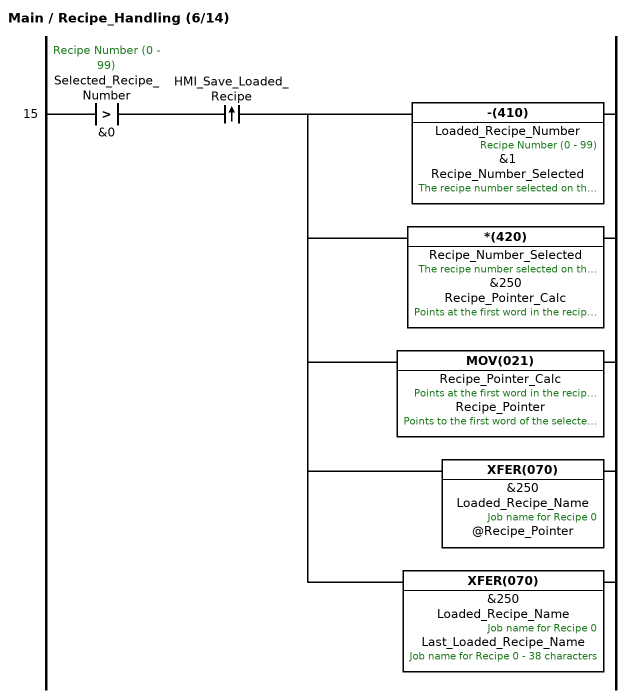
; rung 15
LD>(320) Selected_Recipe_Number &0  ; Recipe Number (0 - 99)
@AND HMI_Save_Loaded_Recipe
-(410) Loaded_Recipe_Number &1 Recipe_Number_Selected  ; Recipe Number (0 - 99), The recipe number selected on the screen.
*(420) Recipe_Number_Selected &250 Recipe_Pointer_Calc  ; The recipe number selected on the screen., Points at the first word in the recipe storage area (E0 - E24999) for the selected recipe.
MOV(021) Recipe_Pointer_Calc Recipe_Pointer  ; Points at the first word in the recipe storage area (E0 - E24999) for the selected recipe., Points to the first word of the selected recipe in the recipe memory area (E0 - E24999)
XFER(070) &250 Loaded_Recipe_Name @Recipe_Pointer  ; Job name for Recipe 0
XFER(070) &250 Loaded_Recipe_Name Last_Loaded_Recipe_Name  ; Job name for Recipe 0, Job name for Recipe 0 - 38 characters

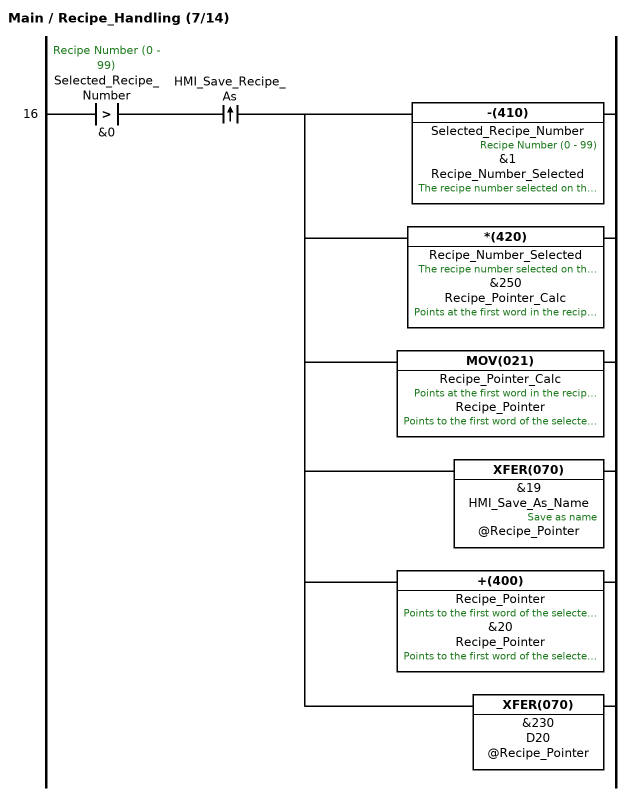
; rung 16
LD>(320) Selected_Recipe_Number &0  ; Recipe Number (0 - 99)
@AND HMI_Save_Recipe_As
-(410) Selected_Recipe_Number &1 Recipe_Number_Selected  ; Recipe Number (0 - 99), The recipe number selected on the screen.
*(420) Recipe_Number_Selected &250 Recipe_Pointer_Calc  ; The recipe number selected on the screen., Points at the first word in the recipe storage area (E0 - E24999) for the selected recipe.
MOV(021) Recipe_Pointer_Calc Recipe_Pointer  ; Points at the first word in the recipe storage area (E0 - E24999) for the selected recipe., Points to the first word of the selected recipe in the recipe memory area (E0 - E24999)
XFER(070) &19 HMI_Save_As_Name @Recipe_Pointer  ; Save as name
+(400) Recipe_Pointer &20 Recipe_Pointer  ; Points to the first word of the selected recipe in the recipe memory area (E0 - E24999)
XFER(070) &230 D20 @Recipe_Pointer

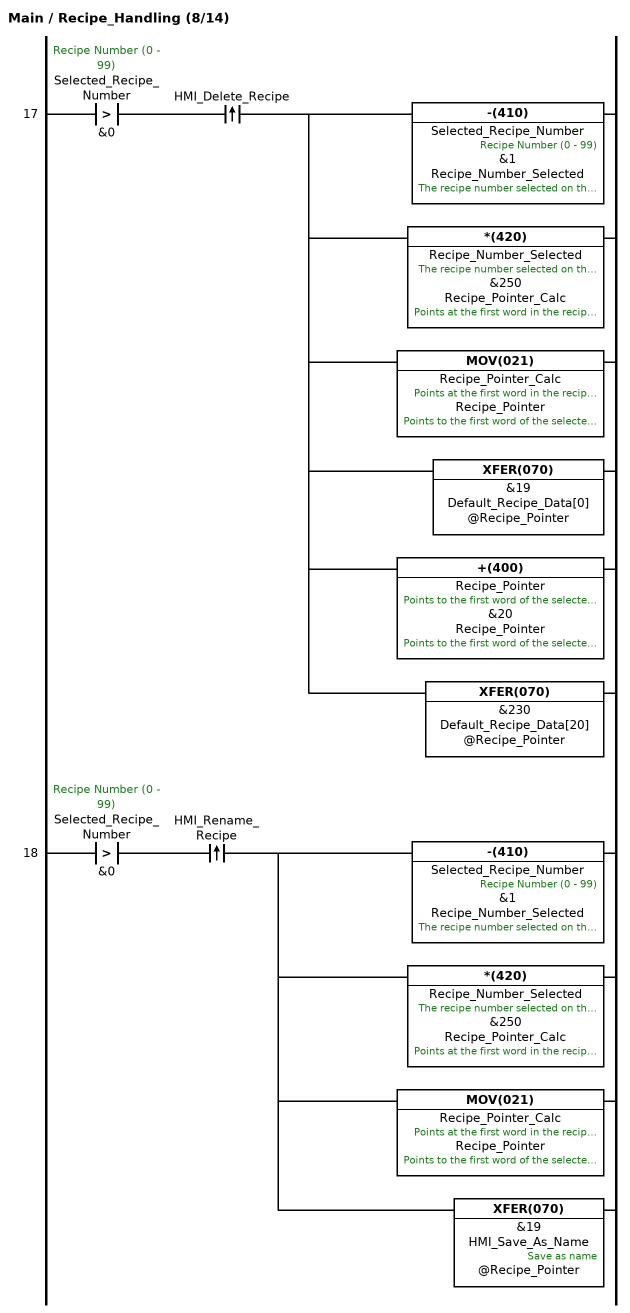
; rung 17
LD>(320) Selected_Recipe_Number &0  ; Recipe Number (0 - 99)
@AND HMI_Delete_Recipe
-(410) Selected_Recipe_Number &1 Recipe_Number_Selected  ; Recipe Number (0 - 99), The recipe number selected on the screen.
*(420) Recipe_Number_Selected &250 Recipe_Pointer_Calc  ; The recipe number selected on the screen., Points at the first word in the recipe storage area (E0 - E24999) for the selected recipe.
MOV(021) Recipe_Pointer_Calc Recipe_Pointer  ; Points at the first word in the recipe storage area (E0 - E24999) for the selected recipe., Points to the first word of the selected recipe in the recipe memory area (E0 - E24999)
XFER(070) &19 Default_Recipe_Data[0] @Recipe_Pointer
+(400) Recipe_Pointer &20 Recipe_Pointer  ; Points to the first word of the selected recipe in the recipe memory area (E0 - E24999)
XFER(070) &230 Default_Recipe_Data[20] @Recipe_Pointer
; rung 18
LD>(320) Selected_Recipe_Number &0  ; Recipe Number (0 - 99)
@AND HMI_Rename_Recipe
-(410) Selected_Recipe_Number &1 Recipe_Number_Selected  ; Recipe Number (0 - 99), The recipe number selected on the screen.
*(420) Recipe_Number_Selected &250 Recipe_Pointer_Calc  ; The recipe number selected on the screen., Points at the first word in the recipe storage area (E0 - E24999) for the selected recipe.
MOV(021) Recipe_Pointer_Calc Recipe_Pointer  ; Points at the first word in the recipe storage area (E0 - E24999) for the selected recipe., Points to the first word of the selected recipe in the recipe memory area (E0 - E24999)
XFER(070) &19 HMI_Save_As_Name @Recipe_Pointer  ; Save as name

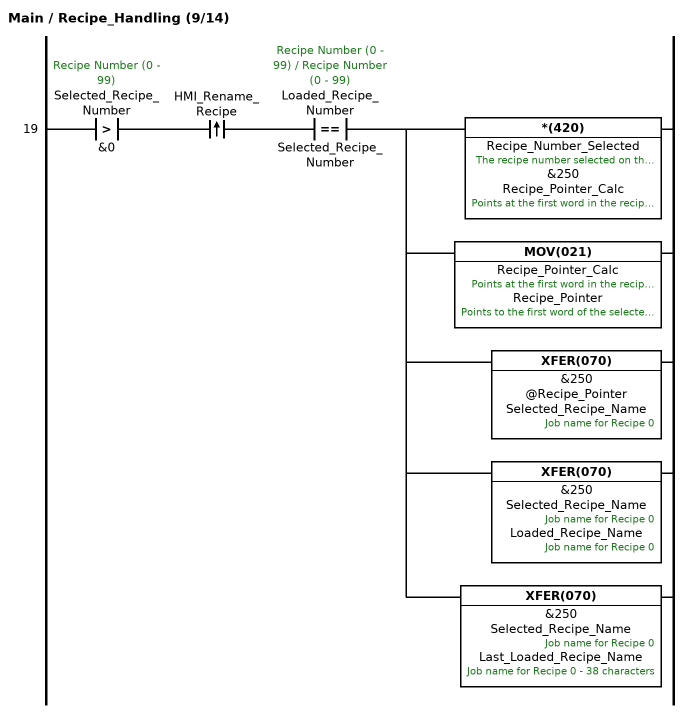
; rung 19
LD>(320) Selected_Recipe_Number &0  ; Recipe Number (0 - 99)
@AND HMI_Rename_Recipe
AND=(300) Loaded_Recipe_Number Selected_Recipe_Number  ; Recipe Number (0 - 99)
*(420) Recipe_Number_Selected &250 Recipe_Pointer_Calc  ; The recipe number selected on the screen., Points at the first word in the recipe storage area (E0 - E24999) for the selected recipe.
MOV(021) Recipe_Pointer_Calc Recipe_Pointer  ; Points at the first word in the recipe storage area (E0 - E24999) for the selected recipe., Points to the first word of the selected recipe in the recipe memory area (E0 - E24999)
XFER(070) &250 @Recipe_Pointer Selected_Recipe_Name  ; Job name for Recipe 0
XFER(070) &250 Selected_Recipe_Name Loaded_Recipe_Name  ; Job name for Recipe 0
XFER(070) &250 Selected_Recipe_Name Last_Loaded_Recipe_Name  ; Job name for Recipe 0, Job name for Recipe 0 - 38 characters

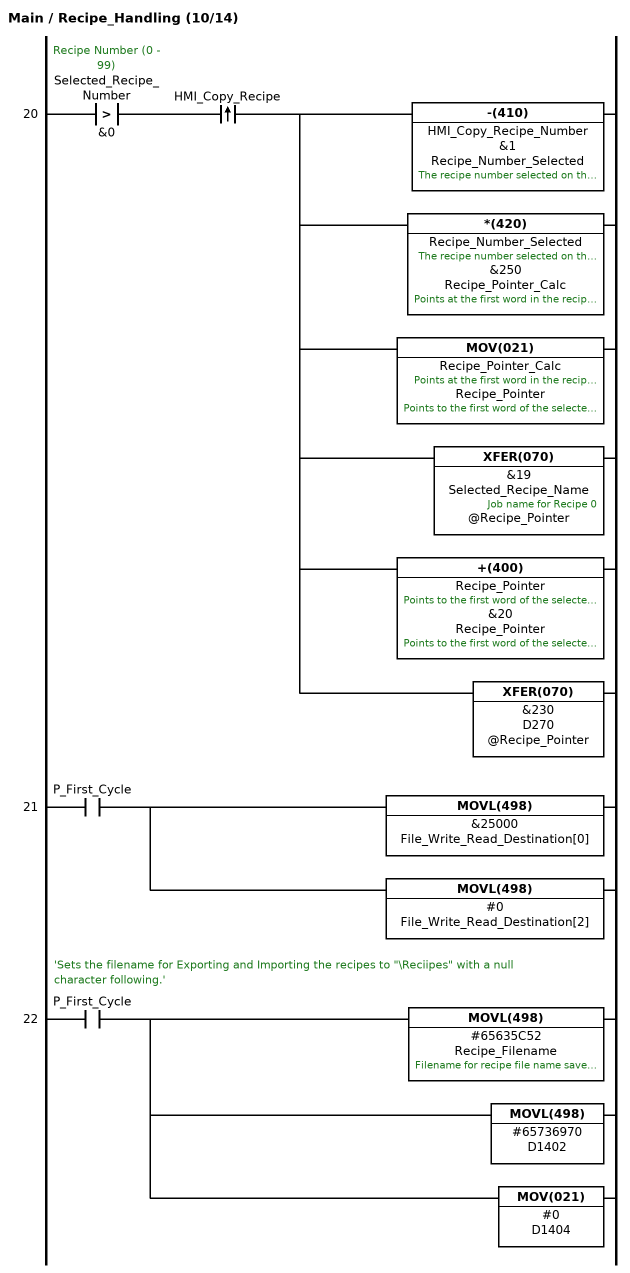
; rung 20
LD>(320) Selected_Recipe_Number &0  ; Recipe Number (0 - 99)
@AND HMI_Copy_Recipe
-(410) HMI_Copy_Recipe_Number &1 Recipe_Number_Selected  ; The recipe number selected on the screen.
*(420) Recipe_Number_Selected &250 Recipe_Pointer_Calc  ; The recipe number selected on the screen., Points at the first word in the recipe storage area (E0 - E24999) for the selected recipe.
MOV(021) Recipe_Pointer_Calc Recipe_Pointer  ; Points at the first word in the recipe storage area (E0 - E24999) for the selected recipe., Points to the first word of the selected recipe in the recipe memory area (E0 - E24999)
XFER(070) &19 Selected_Recipe_Name @Recipe_Pointer  ; Job name for Recipe 0
+(400) Recipe_Pointer &20 Recipe_Pointer  ; Points to the first word of the selected recipe in the recipe memory area (E0 - E24999)
XFER(070) &230 D270 @Recipe_Pointer
; rung 21
LD P_First_Cycle
MOVL(498) &25000 File_Write_Read_Destination[0]  // Sets the number of words to Read / Write to 25000.
MOVL(498) #0 File_Write_Read_Destination[2]  // Sets the offset starting position within the read / write file to 0.
; rung 22: 'Sets the filename for Exporting and Importing the recipes to "\Reciipes" with a null character following.'
LD P_First_Cycle
MOVL(498) #65635C52 Recipe_Filename  ; Filename for recipe file name saved to Compact flash in CSV format
MOVL(498) #65736970 D1402
MOV(021) #0 D1404

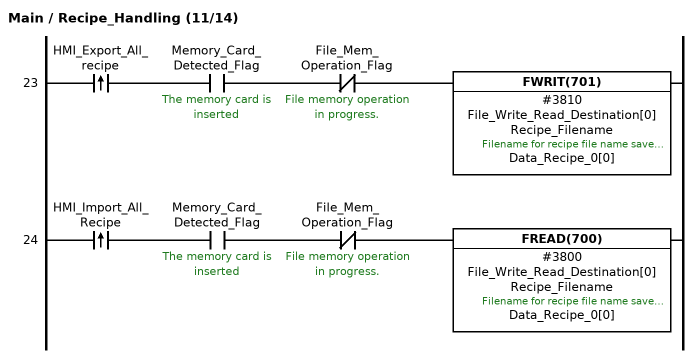
; rung 23
@LD HMI_Export_All_recipe
AND Memory_Card_Detected_Flag  ; The memory card is inserted
ANDNOT File_Mem_Operation_Flag  ; File memory operation in progress.
FWRIT(701) #3810 File_Write_Read_Destination[0] Recipe_Filename Data_Recipe_0[0]  ; Filename for recipe file name saved to Compact flash in CSV format
; rung 24
@LD HMI_Import_All_Recipe
AND Memory_Card_Detected_Flag  ; The memory card is inserted
ANDNOT File_Mem_Operation_Flag  ; File memory operation in progress.
FREAD(700) #3800 File_Write_Read_Destination[0] Recipe_Filename Data_Recipe_0[0]  ; Filename for recipe file name saved to Compact flash in CSV format

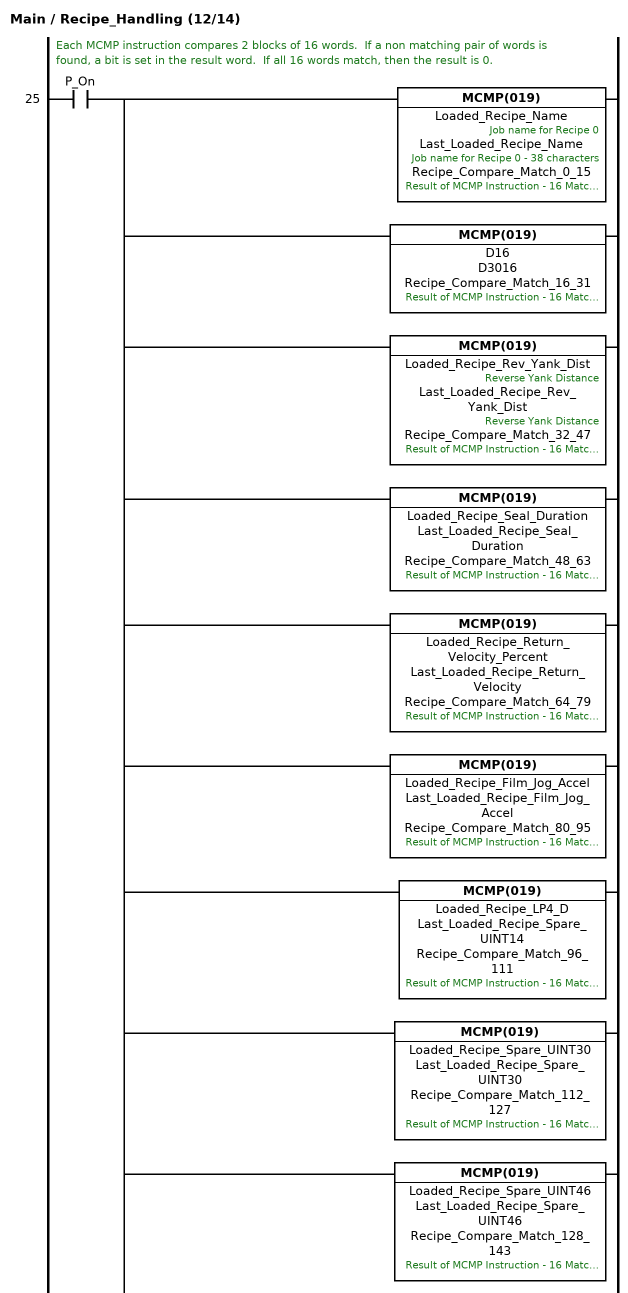

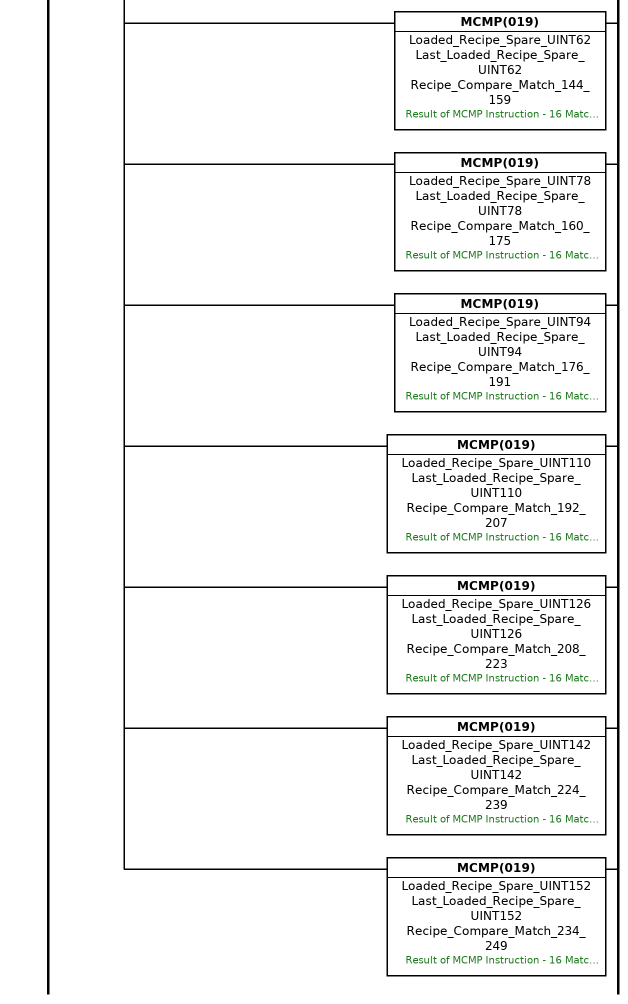
; rung 25: Each MCMP instruction compares 2 blocks of 16 words.  If a non matching pair of words is found, a bit is set in the result word.  If all 16 words match, then the result is 0.
LD P_On
MCMP(019) Loaded_Recipe_Name Last_Loaded_Recipe_Name Recipe_Compare_Match_0_15  ; Job name for Recipe 0, Job name for Recipe 0 - 38 characters, Result of MCMP Instruction - 16 Match Conditions
MCMP(019) D16 D3016 Recipe_Compare_Match_16_31  ; Result of MCMP Instruction - 16 Match Conditions
MCMP(019) Loaded_Recipe_Rev_Yank_Dist Last_Loaded_Recipe_Rev_Yank_Dist Recipe_Compare_Match_32_47  ; Reverse Yank Distance, Result of MCMP Instruction - 16 Match Conditions
MCMP(019) Loaded_Recipe_Seal_Duration Last_Loaded_Recipe_Seal_Duration Recipe_Compare_Match_48_63  ; Result of MCMP Instruction - 16 Match Conditions
MCMP(019) Loaded_Recipe_Return_Velocity_Percent Last_Loaded_Recipe_Return_Velocity Recipe_Compare_Match_64_79  ; Result of MCMP Instruction - 16 Match Conditions
MCMP(019) Loaded_Recipe_Film_Jog_Accel Last_Loaded_Recipe_Film_Jog_Accel Recipe_Compare_Match_80_95  ; Result of MCMP Instruction - 16 Match Conditions
MCMP(019) Loaded_Recipe_LP4_D Last_Loaded_Recipe_Spare_UINT14 Recipe_Compare_Match_96_111  ; Result of MCMP Instruction - 16 Match Conditions
MCMP(019) Loaded_Recipe_Spare_UINT30 Last_Loaded_Recipe_Spare_UINT30 Recipe_Compare_Match_112_127  ; Result of MCMP Instruction - 16 Match Conditions
MCMP(019) Loaded_Recipe_Spare_UINT46 Last_Loaded_Recipe_Spare_UINT46 Recipe_Compare_Match_128_143  ; Result of MCMP Instruction - 16 Match Conditions
MCMP(019) Loaded_Recipe_Spare_UINT62 Last_Loaded_Recipe_Spare_UINT62 Recipe_Compare_Match_144_159  ; Result of MCMP Instruction - 16 Match Conditions
MCMP(019) Loaded_Recipe_Spare_UINT78 Last_Loaded_Recipe_Spare_UINT78 Recipe_Compare_Match_160_175  ; Result of MCMP Instruction - 16 Match Conditions
MCMP(019) Loaded_Recipe_Spare_UINT94 Last_Loaded_Recipe_Spare_UINT94 Recipe_Compare_Match_176_191  ; Result of MCMP Instruction - 16 Match Conditions
MCMP(019) Loaded_Recipe_Spare_UINT110 Last_Loaded_Recipe_Spare_UINT110 Recipe_Compare_Match_192_207  ; Result of MCMP Instruction - 16 Match Conditions
MCMP(019) Loaded_Recipe_Spare_UINT126 Last_Loaded_Recipe_Spare_UINT126 Recipe_Compare_Match_208_223  ; Result of MCMP Instruction - 16 Match Conditions
MCMP(019) Loaded_Recipe_Spare_UINT142 Last_Loaded_Recipe_Spare_UINT142 Recipe_Compare_Match_224_239  ; Result of MCMP Instruction - 16 Match Conditions
MCMP(019) Loaded_Recipe_Spare_UINT152 Last_Loaded_Recipe_Spare_UINT152 Recipe_Compare_Match_234_249  ; Result of MCMP Instruction - 16 Match Conditions - Overlap with previouis to end right at 249  // This instruction overlaps with the previous to end the comparisons right at 249.

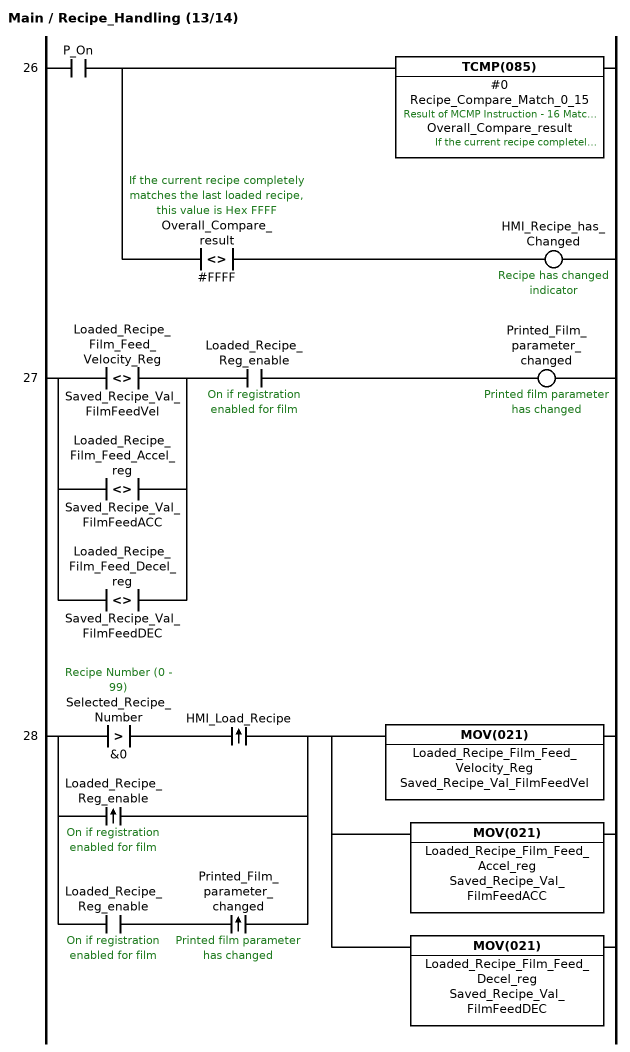
; rung 26
LD P_On
TCMP(085) #0 Recipe_Compare_Match_0_15 Overall_Compare_result  ; Result of MCMP Instruction - 16 Match Conditions, If the current recipe completely matches the last loaded recipe, this value is Hex FFFF
AND<>(305) Overall_Compare_result #FFFF  ; If the current recipe completely matches the last loaded recipe, this value is Hex FFFF
OUT HMI_Recipe_has_Changed  ; Recipe has changed indicator
; rung 27
LD<>(305) Loaded_Recipe_Film_Feed_Velocity_Reg Saved_Recipe_Val_FilmFeedVel
OR<>(305) Loaded_Recipe_Film_Feed_Accel_reg Saved_Recipe_Val_FilmFeedACC
OR<>(305) Loaded_Recipe_Film_Feed_Decel_reg Saved_Recipe_Val_FilmFeedDEC
AND Loaded_Recipe_Reg_enable  ; On if registration enabled for film
OUT Printed_Film_parameter_changed  ; Printed film parameter has changed
; rung 28
LD>(320) Selected_Recipe_Number &0  ; Recipe Number (0 - 99)
@AND HMI_Load_Recipe
@OR Loaded_Recipe_Reg_enable  ; On if registration enabled for film
LD Loaded_Recipe_Reg_enable  ; On if registration enabled for film
@AND Printed_Film_parameter_changed  ; Printed film parameter has changed
ORLD
MOV(021) Loaded_Recipe_Film_Feed_Velocity_Reg Saved_Recipe_Val_FilmFeedVel
MOV(021) Loaded_Recipe_Film_Feed_Accel_reg Saved_Recipe_Val_FilmFeedACC
MOV(021) Loaded_Recipe_Film_Feed_Decel_reg Saved_Recipe_Val_FilmFeedDEC

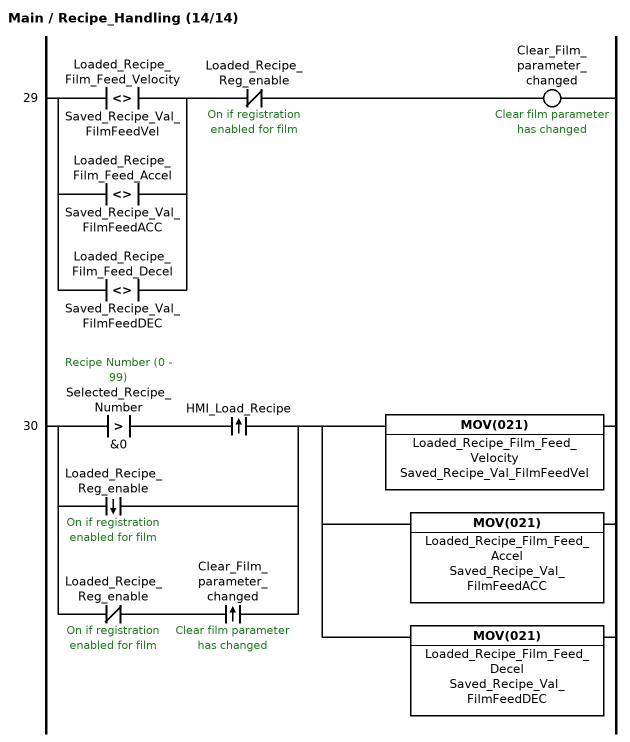
; rung 29
LD<>(305) Loaded_Recipe_Film_Feed_Velocity Saved_Recipe_Val_FilmFeedVel
OR<>(305) Loaded_Recipe_Film_Feed_Accel Saved_Recipe_Val_FilmFeedACC
OR<>(305) Loaded_Recipe_Film_Feed_Decel Saved_Recipe_Val_FilmFeedDEC
ANDNOT Loaded_Recipe_Reg_enable  ; On if registration enabled for film
OUT Clear_Film_parameter_changed  ; Clear film parameter has changed
; rung 30
LD>(320) Selected_Recipe_Number &0  ; Recipe Number (0 - 99)
@AND HMI_Load_Recipe
%OR Loaded_Recipe_Reg_enable  ; On if registration enabled for film
LDNOT Loaded_Recipe_Reg_enable  ; On if registration enabled for film
@AND Clear_Film_parameter_changed  ; Clear film parameter has changed
ORLD
MOV(021) Loaded_Recipe_Film_Feed_Velocity Saved_Recipe_Val_FilmFeedVel
MOV(021) Loaded_Recipe_Film_Feed_Accel Saved_Recipe_Val_FilmFeedACC
MOV(021) Loaded_Recipe_Film_Feed_Decel Saved_Recipe_Val_FilmFeedDEC

### Section Overal_Machine

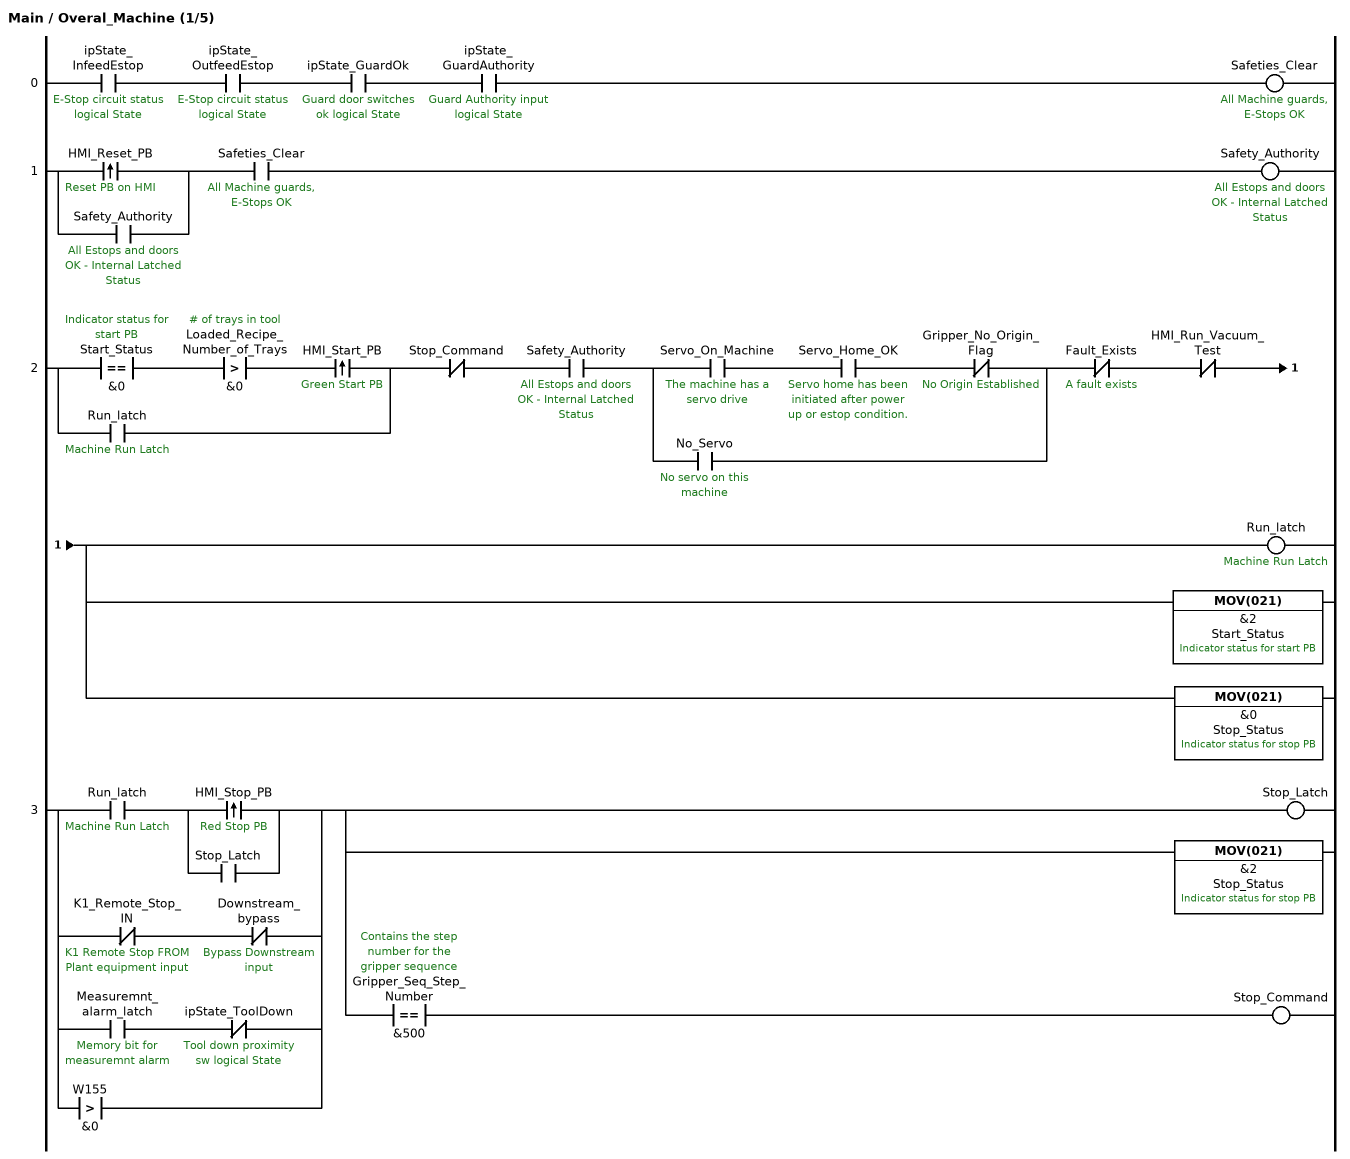
; rung 0
LD ipState_InfeedEstop  ; E-Stop circuit status logical State
AND ipState_OutfeedEstop  ; E-Stop circuit status logical State
AND ipState_GuardOk  ; Guard door switches ok logical State
AND ipState_GuardAuthority  ; Guard Authority input logical State
OUT Safeties_Clear  ; All Machine guards, E-Stops OK
; rung 1
@LD HMI_Reset_PB  ; Reset PB on HMI
OR Safety_Authority  ; All Estops and doors OK - Internal Latched Status
AND Safeties_Clear  ; All Machine guards, E-Stops OK
OUT Safety_Authority  ; All Estops and doors OK - Internal Latched Status
; rung 2
LD=(300) Start_Status &0  ; Indicator status for start PB
AND>(320) Loaded_Recipe_Number_of_Trays &0  ; # of trays in tool
@AND HMI_Start_PB  ; Green Start PB
OR Run_latch  ; Machine Run Latch
ANDNOT Stop_Command
AND Safety_Authority  ; All Estops and doors OK - Internal Latched Status
LD Servo_On_Machine  ; The machine has a servo drive
AND Servo_Home_OK  ; Servo home has been initiated after power up or estop condition.
ANDNOT Gripper_No_Origin_Flag  ; No Origin Established
OR No_Servo  ; No servo on this machine
ANDLD
ANDNOT Fault_Exists  ; A fault exists
ANDNOT HMI_Run_Vacuum_Test
OUT Run_latch  ; Machine Run Latch
MOV(021) &2 Start_Status  ; Indicator status for start PB
MOV(021) &0 Stop_Status  ; Indicator status for stop PB
; rung 3
LD Run_latch  ; Machine Run Latch
@LD HMI_Stop_PB  ; Red Stop PB
OR Stop_Latch
ANDLD
LDNOT K1_Remote_Stop_IN  ; K1 Remote Stop FROM Plant equipment input
ANDNOT Downstream_bypass  ; Bypass Downstream input
ORLD
LD Measuremnt_alarm_latch  ; Memory bit for measuremnt alarm
ANDNOT ipState_ToolDown  ; Tool down proximity sw logical State
ORLD
OR>(320) W155 &0
OUT Stop_Latch
MOV(021) &2 Stop_Status  ; Indicator status for stop PB
AND=(300) Gripper_Seq_Step_Number &500  ; Contains the step number for the gripper sequence
OUT Stop_Command

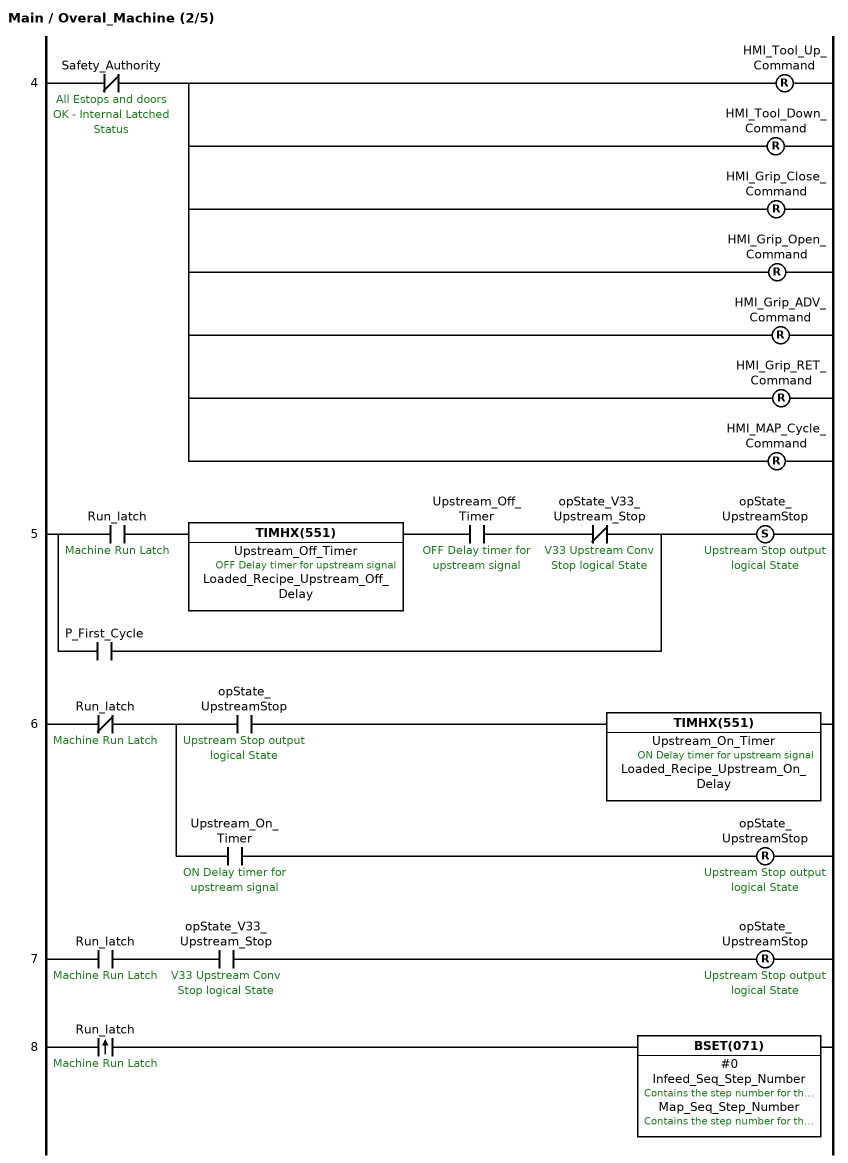
; rung 4
LDNOT Safety_Authority  ; All Estops and doors OK - Internal Latched Status
RSET HMI_Tool_Up_Command
RSET HMI_Tool_Down_Command
RSET HMI_Grip_Close_Command
RSET HMI_Grip_Open_Command
RSET HMI_Grip_ADV_Command
RSET HMI_Grip_RET_Command
RSET HMI_MAP_Cycle_Command
; rung 5
LD Run_latch  ; Machine Run Latch
TIMHX(551) Upstream_Off_Timer Loaded_Recipe_Upstream_Off_Delay  ; OFF Delay timer for upstream signal
AND Upstream_Off_Timer  ; OFF Delay timer for upstream signal
ANDNOT opState_V33_Upstream_Stop  ; V33 Upstream Conv Stop logical State
OR P_First_Cycle
SET opState_UpstreamStop  ; Upstream Stop output logical State
; rung 6
LDNOT Run_latch  ; Machine Run Latch
OUT TR0
AND opState_UpstreamStop  ; Upstream Stop output logical State
TIMHX(551) Upstream_On_Timer Loaded_Recipe_Upstream_On_Delay  ; ON Delay timer for upstream signal
LD TR0
AND Upstream_On_Timer  ; ON Delay timer for upstream signal
RSET opState_UpstreamStop  ; Upstream Stop output logical State
; rung 7
LD Run_latch  ; Machine Run Latch
AND opState_V33_Upstream_Stop  ; V33 Upstream Conv Stop logical State
RSET opState_UpstreamStop  ; Upstream Stop output logical State
; rung 8
@LD Run_latch  ; Machine Run Latch
BSET(071) #0 Infeed_Seq_Step_Number Map_Seq_Step_Number  ; Contains the step number for the Infeed sequence, Contains the step number for the map sequence

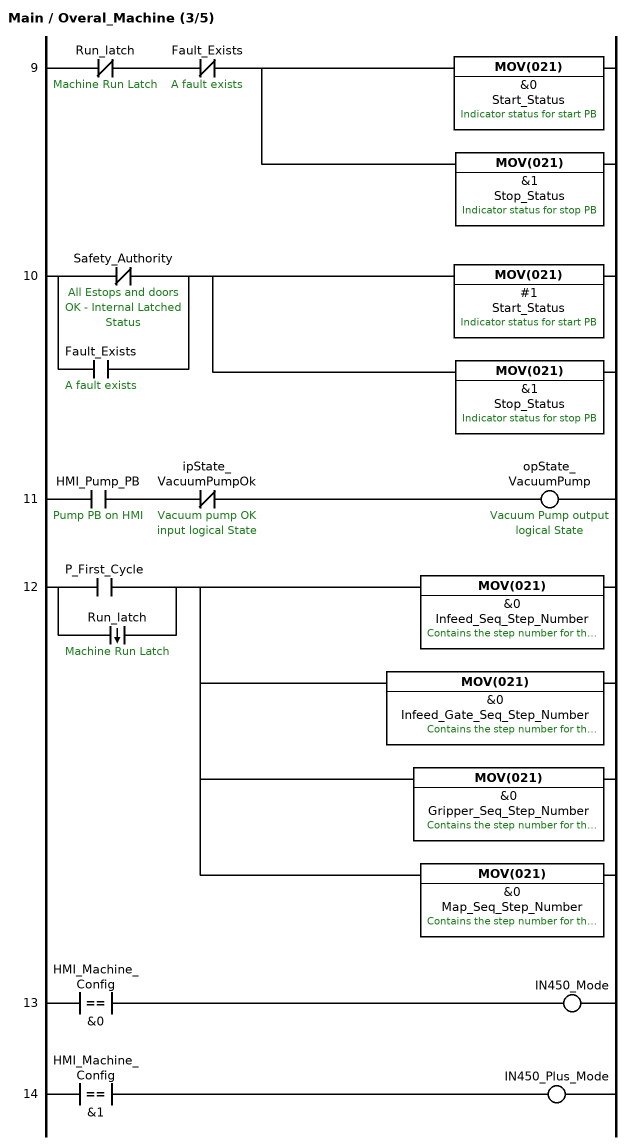
; rung 9
LDNOT Run_latch  ; Machine Run Latch
ANDNOT Fault_Exists  ; A fault exists
MOV(021) &0 Start_Status  ; Indicator status for start PB
MOV(021) &1 Stop_Status  ; Indicator status for stop PB
; rung 10
LDNOT Safety_Authority  ; All Estops and doors OK - Internal Latched Status
OR Fault_Exists  ; A fault exists
MOV(021) #1 Start_Status  ; Indicator status for start PB
MOV(021) &1 Stop_Status  ; Indicator status for stop PB
; rung 11
LD HMI_Pump_PB  ; Pump PB on HMI
ANDNOT ipState_VacuumPumpOk  ; Vacuum pump OK input logical State
OUT opState_VacuumPump  ; Vacuum Pump output logical State
; rung 12
LD P_First_Cycle
%OR Run_latch  ; Machine Run Latch
MOV(021) &0 Infeed_Seq_Step_Number  ; Contains the step number for the Infeed sequence
MOV(021) &0 Infeed_Gate_Seq_Step_Number  ; Contains the step number for the infeed gate sequence
MOV(021) &0 Gripper_Seq_Step_Number  ; Contains the step number for the gripper sequence
MOV(021) &0 Map_Seq_Step_Number  ; Contains the step number for the map sequence
; rung 13
LD=(300) HMI_Machine_Config &0
OUT IN450_Mode
; rung 14
LD=(300) HMI_Machine_Config &1
OUT IN450_Plus_Mode

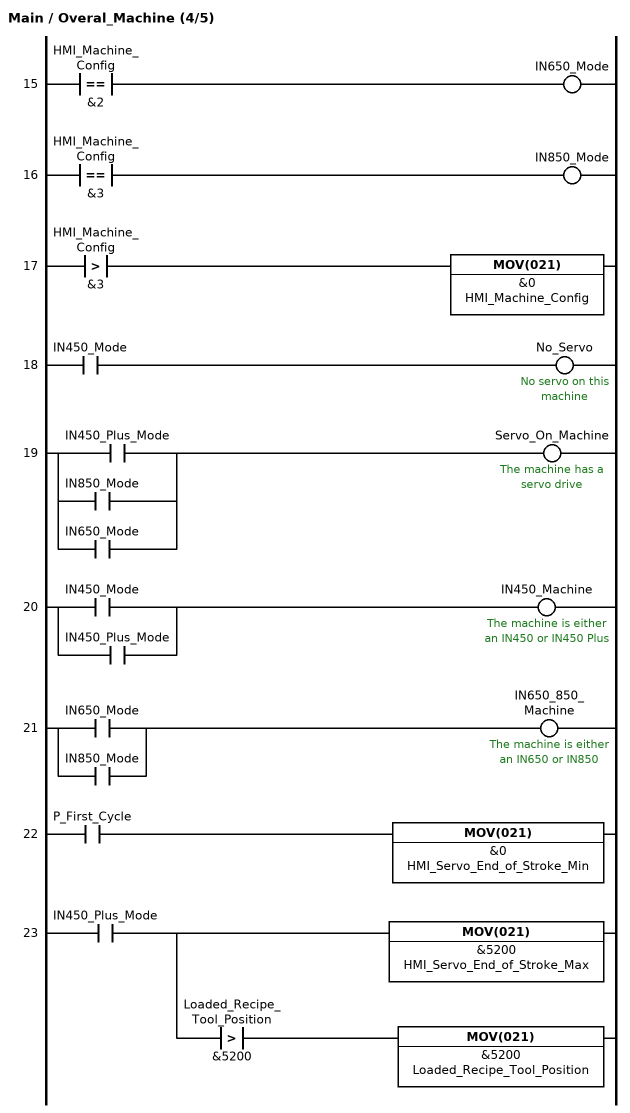
; rung 15
LD=(300) HMI_Machine_Config &2
OUT IN650_Mode
; rung 16
LD=(300) HMI_Machine_Config &3
OUT IN850_Mode
; rung 17
LD>(320) HMI_Machine_Config &3
MOV(021) &0 HMI_Machine_Config
; rung 18
LD IN450_Mode
OUT No_Servo  ; No servo on this machine
; rung 19
LD IN450_Plus_Mode
OR IN850_Mode
OR IN650_Mode
OUT Servo_On_Machine  ; The machine has a servo drive
; rung 20
LD IN450_Mode
OR IN450_Plus_Mode
OUT IN450_Machine  ; The machine is either an IN450 or IN450 Plus
; rung 21
LD IN650_Mode
OR IN850_Mode
OUT IN650_850_Machine  ; The machine is either an IN650 or IN850
; rung 22
LD P_First_Cycle
MOV(021) &0 HMI_Servo_End_of_Stroke_Min
; rung 23
LD IN450_Plus_Mode
MOV(021) &5200 HMI_Servo_End_of_Stroke_Max
AND>(320) Loaded_Recipe_Tool_Position &5200
MOV(021) &5200 Loaded_Recipe_Tool_Position

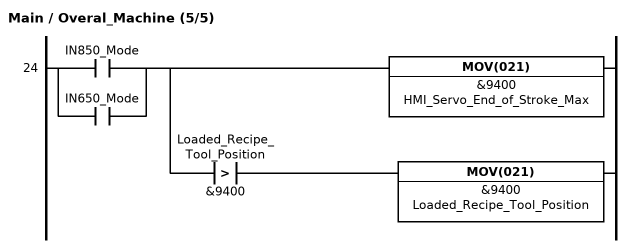
; rung 24
LD IN850_Mode
OR IN650_Mode
MOV(021) &9400 HMI_Servo_End_of_Stroke_Max
AND>(320) Loaded_Recipe_Tool_Position &9400
MOV(021) &9400 Loaded_Recipe_Tool_Position

### Section Infeed_Sequence

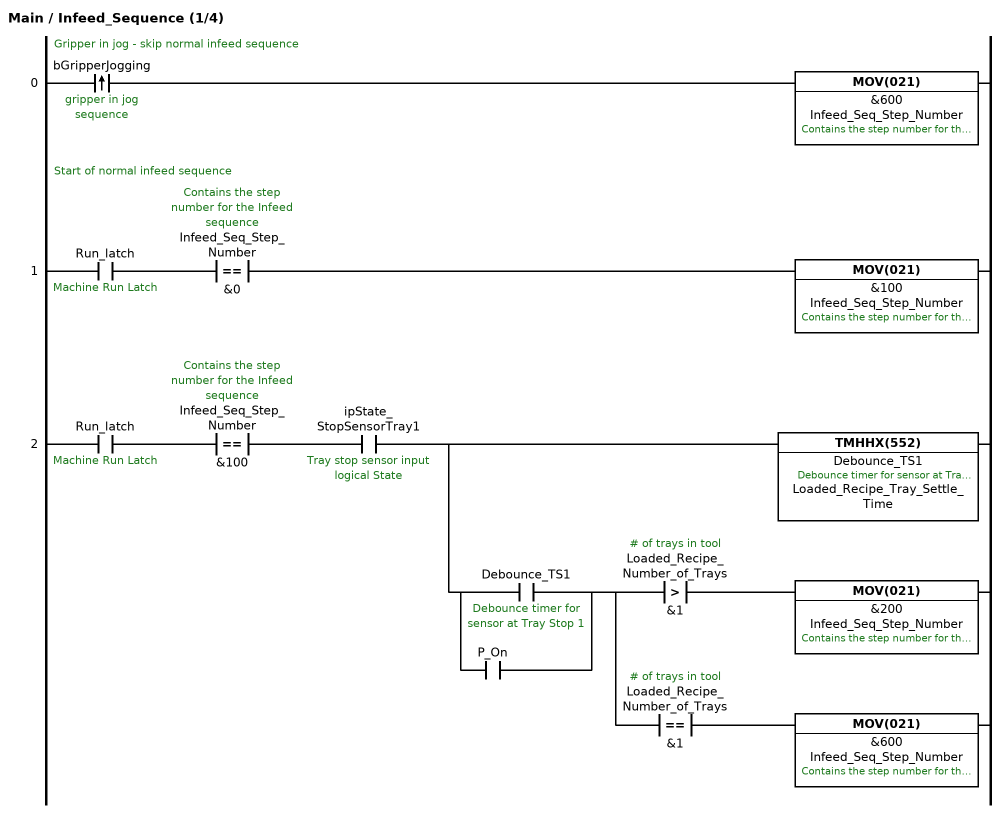
; rung 0: Gripper in jog - skip normal infeed sequence
@LD bGripperJogging  ; gripper in jog sequence
MOV(021) &600 Infeed_Seq_Step_Number  ; Contains the step number for the Infeed sequence
; rung 1: Start of normal infeed sequence
LD Run_latch  ; Machine Run Latch
AND=(300) Infeed_Seq_Step_Number &0  ; Contains the step number for the Infeed sequence
MOV(021) &100 Infeed_Seq_Step_Number  ; Contains the step number for the Infeed sequence
; rung 2
LD Run_latch  ; Machine Run Latch
AND=(300) Infeed_Seq_Step_Number &100  ; Contains the step number for the Infeed sequence
AND ipState_StopSensorTray1  ; Tray stop sensor input logical State
TMHHX(552) Debounce_TS1 Loaded_Recipe_Tray_Settle_Time  ; Debounce timer for sensor at Tray Stop 1
LD Debounce_TS1  ; Debounce timer for sensor at Tray Stop 1
OR P_On  // Sensor on and off filters added elsewhere.  Bypassed on 9/25/14 per Gary Liles.
ANDLD
OUT TR0
AND>(320) Loaded_Recipe_Number_of_Trays &1  ; # of trays in tool
MOV(021) &200 Infeed_Seq_Step_Number  ; Contains the step number for the Infeed sequence
LD TR0
AND=(300) Loaded_Recipe_Number_of_Trays &1  ; # of trays in tool
MOV(021) &600 Infeed_Seq_Step_Number  ; Contains the step number for the Infeed sequence

